// TIA Portal project "9230A V00 - PI" (V16)

(* hardware
DEVICE "S7-1200 station_1"  S7-1200 Station
   slot 0: "Rack_0"  S7-1200 Rack  Rack  V1.0
   slot 1: "1U2"  CPU 1212C DC/DC/DC  6ES7 212-1AE40-0XB0  V4.4
   slot 2: "2U2"  SM 1222 DQ8 x 24VDC  6ES7 222-1BF32-0XB0  V2.0
DEVICE "GSD device_1"  GSD.Device.PN
   slot 0: "Rack"  Rack  V1.0
   slot 0: "8DI"  8DI
   slot 0: "8DO"  8DO
   slot 0: "8DO"  8DO
   slot 0: "4AI, INT16[4] I"  4AI, INT16[4] I
   slot 0: "1U1"  750-375 V02.05.xx (FW 08)  750-375  V02.05.xx (08)
      slot 0: "Big Endian (MOTOROLA), Subslot-controlled PROFIenergy"  Big Endian (MOTOROLA), Subslot-controlled PROFIenergy
      slot 1: "Interface"  Interface
         slot 1: "Port 1"  Port 1
         slot 2: "Port 2"  Port 2
   slot 1: "2U1"  75x-430(/0..-...) 8DI  75x-430
   slot 2: "3U1"  75x-530(/0..-...) 8DO  75x-530
   slot 3: "4U1"  75x-530(/0..-...) 8DO  75x-530
   slot 4: "5U1"  75x-455(/0..-000) 4AI 4-20 mA s.e.  75x-455(/0..-000)
DEVICE "GSD device_2"  GSD.Device.PN
   slot 0: "Rack"  Rack  V1.0
   slot 0: "4AI, INT16[4] I"  4AI, INT16[4] I
   slot 0: "8DI"  8DI
   slot 0: "8DO"  8DO
   slot 0: "1U3"  750-375 V02.05.xx (FW 08)  750-375  V02.05.xx (08)
      slot 0: "Big Endian (MOTOROLA), Subslot-controlled PROFIenergy"  Big Endian (MOTOROLA), Subslot-controlled PROFIenergy
      slot 1: "Interface"  Interface
         slot 1: "Port 1"  Port 1
         slot 2: "Port 2"  Port 2
   slot 1: "2U3"  75x-430(/0..-...) 8DI  75x-430
   slot 2: "3U3"  75x-530(/0..-...) 8DO  75x-530
   slot 3: "4U3"  75x-455(/0..-000) 4AI 4-20 mA s.e.  75x-455(/0..-000)
DEVICE "SINAMICS G_1"  Sinamics.Device
   slot 0: "	_0"  Rail  SinamicsG120CRackP
   slot 0: "43G1"  G120C PN  6SL3210-1KE12-3UF2  4.7.10
      slot 1: "PROFINET interface"  MDD-SinamicsG120-P
      slot 3: "PM G120C"  PM G120C  6SL3210-1KE12-3UF2  -
DEVICE "SINAMICS G_2"  Sinamics.Device
   slot 0: "	_0"  Rail  SinamicsG120CRackP
   slot 0: "62G1"  G120C PN  6SL3210-1KE14-3UF2  4.7.10
      slot 1: "PROFINET interface"  MDD-SinamicsG120-P
      slot 3: "PM G120C"  PM G120C  6SL3210-1KE14-3UF2  -
DEVICE "SINAMICS G_3"  Sinamics.Device
   slot 0: "	_0"  Rail  SinamicsG120CRackP
   slot 0: "65G1"  G120C PN  6SL3210-1KE15-8UF2  4.7.10
      slot 1: "PROFINET interface"  MDD-SinamicsG120-P
      slot 3: "PM G120C"  PM G120C  6SL3210-1KE15-8UF2  -
DEVICE "SCALANCE X005"  SCALANCE X-Station
   slot 0: "SCALANCE X rack"  Rail
   slot 0: "Switch"  6GK5 008-0BA10-1AB2  V1.0
*)

// ===== PLC "1U2"  CPU 1212C DC/DC/DC =====

VAR_GLOBAL   // PLC tag table "Default tag table"
   "System_Byte" AT %MB1 : Byte;
   "FirstScan" AT %M1.0 : Bool;
   "DiagStatusUpdate" AT %M1.1 : Bool;
   "AlwaysTRUE" AT %M1.2 : Bool;
   "AlwaysFALSE" AT %M1.3 : Bool;
   "Clock_10Hz" AT %M0.0 : Bool;
   "Clock_5Hz" AT %M0.1 : Bool;
   "Clock_2.5Hz" AT %M0.2 : Bool;
   "Clock_2Hz" AT %M0.3 : Bool;
   "Clock_1.25Hz" AT %M0.4 : Bool;
   "Clock_1Hz" AT %M0.5 : Bool;
   "Clock_0.625Hz" AT %M0.6 : Bool;
   "Clock_0.5Hz" AT %M0.7 : Bool;
   "Clock_Byte" AT %MB0 : Byte;
   "Emergencia_Painel_1" AT %M7.5 : Bool;
   "Emergencia_Painel_3" AT %M7.6 : Bool;
   "Emergencia_Painel_2" AT %M7.7 : Bool;
END_VAR

VAR_GLOBAL   // PLC tag table "IO PAINEL 1"
   "EMERGENCIA_GERAL_PAINEL_1" AT %I1.0 : Bool;
   "NIVEL_SUPERIOR_SILO_2" AT %I1.1 : Bool;
   "SENSOR_23_POSICAO_1" AT %I1.2 : Bool;
   "NIVEL_INFERIOR_SILO_1" AT %I1.3 : Bool;
   "NIVEL_INFERIOR_SILO_2" AT %I1.5 : Bool;
   "SENSOR_23_POSICAO_2" AT %I1.4 : Bool;
   "NIVEL_SUPERIOR_SILO_1" AT %I1.6 : Bool;
   "BT_27_DOSAGEM_MANUAL" AT %I1.7 : Bool;
   "LIGA_LED_BT_27_DOSAGEM_MANUAL" AT %Q1.1 : Bool;
   "LIGA_22" AT %Q1.2 : Bool;
   "LIGA_26_SILO1_SENTIDO_1" AT %Q1.3 : Bool;
   "LIGA_23_SENTIDO_1" AT %Q1.4 : Bool;
   "LIGA_26_SILO1_SENTIDO_2" AT %Q1.5 : Bool;
   "LIGA_23_SENTIDO_2" AT %Q1.6 : Bool;
   "LIGA_26_SILO2_SENTIDO_1" AT %Q1.7 : Bool;
   "LIGA_26_SILO2_SENTIDO_2" AT %Q2.0 : Bool;
   "TARA_BALANCA_DOSAGEM" AT %Q2.1 : Bool;
   "LIGA_29" AT %Q2.2 : Bool;
   "LIGA_30" AT %Q2.4 : Bool;
   "ZERO_BALANCA_DOSAGEM" AT %Q2.6 : Bool;
   "POSICAO_ATUAL_26_SILO1" AT %IW68 : Int;
   "POSICAO_ATUAL_26_SILO2" AT %IW72 : Int;
   "PESO_ATUAL_DOSAGEM" AT %IW70 : Int;
END_VAR

VAR_GLOBAL   // PLC tag table "IO PAINEL 2"
   "LIGA_48" AT %Q8.0 : Bool;
   "LIGA_49_SENTIDO_1" AT %Q8.1 : Bool;
   "LIGA_49_SENTIDO_2" AT %Q8.2 : Bool;
   "CORRENTE_ATUAL_44" AT %IW64 : Int;
   "EMERGENCIA_GERAL_PAINEL_2" AT %I0.0 : Bool;
   "FALTA_FASE" AT %I0.1 : Bool;
   "NIVEL_INFERIOR_PRE_MISTURADOR" AT %I0.2 : Bool;
   "NIVEL_INFERIOR_POS_MISTURADOR" AT %I0.3 : Bool;
   "SENSOR_49_SENTIDO_1" AT %I0.4 : Bool;
   "SENSOR_49_SENTIDO_2" AT %I0.5 : Bool;
   "LIGA_42" AT %Q0.0 : Bool;
   "LIGA_CONTATOR_1_44" AT %Q0.1 : Bool;
   "LIGA_CONTATOR_2_44" AT %Q0.2 : Bool;
   "LIGA_44" AT %Q0.3 : Bool;
   "LIGA_45" AT %Q0.4 : Bool;
   "LIGA_46" AT %Q0.5 : Bool;
END_VAR

VAR_GLOBAL   // PLC tag table "IO PAINEL 3"
   "PESO_ATUAL_ENSAQUE" AT %IW76 : Int;
   "TARA_BALANCA_ENSAQUE" AT %Q3.2 : Bool;
   "ZERO_BALANCA_ENSAQUE" AT %Q3.0 : Bool;
   "EMERGENCIA_GERAL_PAINEL_3" AT %I2.0 : Bool;
   "NIVEL_SUPERIOR_SILO_EXP" AT %I2.2 : Bool;
   "NIVEL_INFERIOR_SILO_EXP" AT %I2.4 : Bool;
   "PEDAL_ENSAQUE" AT %I2.6 : Bool;
END_VAR

VAR_GLOBAL   // PLC tag table "teste"
   "TESTE" AT %MW16 : Int;
   "TESTE1" AT %MD12 : Real;
   "TESTE2" AT %MD8 : Real;
   "TESTE3" AT %M6.0 : Bool;
   "TESTE33" AT %MD2 : Real;
   "teste22" AT %MD18 : Real;
   "teste333" AT %MD22 : Real;
   "teste444" AT %MD26 : Real;
   "teste55" AT %MD30 : Real;
   "teste66" AT %M6.1 : Bool;
   "teste777" AT %M6.2 : Bool;
   "asdff" AT %M6.3 : Bool;
   "fdvxc" AT %M6.4 : Bool;
   "nhgfbvdc" AT %M6.5 : Bool;
   "teste123" AT %M6.7 : Bool;
   "tesdfsfdg" AT %M6.6 : Bool;
   "sdfvxc" AT %M7.0 : Bool;
   "teste88" AT %M7.1 : Bool;
   "teste99" AT %M7.2 : Bool;
   "teste00" AT %M7.3 : Bool;
   "teste3333" AT %M7.4 : Bool;
   "teste11" AT %M34.0 : Bool;
   "teste12" AT %M34.1 : Bool;
   "teste13" AT %M34.2 : Bool;
   "dfdfgsfgd" AT %M34.3 : Bool;
   "hngfnbfgn" AT %M34.4 : Bool;
   "teste411" AT %M34.5 : Bool;
   "teste412" AT %M34.6 : Bool;
END_VAR

TYPE "typeAtuadorLinearDigital"
   STRUCT
      Manual : Bool;   // em manual
      Automatico : Bool;   // em automatico
      Manutencao : Bool;   // em manutencao
      Libera_Bloqueio_Manual : Bool;   // Libera Bloqueio do motor
      Em_Emergencia : Bool;   // Em emergencia
      Liberado : Bool;   // Liberado
      Aciona_Lado1 : Bool;   // Comando aciona Lado
      Aciona_Lado2 : Bool;   // Comando aciona Lado
      Acionando_Lado1 : Bool;   // status acionando lado
      Acionando_Lado2 : Bool;   // status acionando lado
      Acionando_Automatico : Bool;   // acionando em modo automatico
      Em_Posicao_Lado1 : Bool;   // status lado atual
      Em_Posicao_Lado2 : Bool;   // status lado atual
      Falha_Acionando_Lado1 : Bool;   // falha acionando lado 1
      Falha_Acionando_Lado2 : Bool;   // falha acionando lado 2
      Falha_2_Posicoes_Ativa : Bool;   // falha quando os dois sensores estiverem ativos
      Falha_Confirmacao_Contator_Lado1 : Bool;   // falha no contator ou fio de confirmação do lado 1
      Falha_Confirmacao_Contator_Lado2 : Bool;   // falha no contator ou fio de confirmação do lado 2
      Reset_Falha : Bool;   // reset falha
      bitReserva : Bool;
      bitReserva_1 : Bool;
      bitReserva_2 : Bool;
      bitReserva_3 : Bool;
      bitReserva_4 : Bool;
      bitReserva_5 : Bool;
      bitReserva_6 : Bool;
      bitReserva_7 : Bool;
      bitReserva_8 : Bool;
      bitReserva_9 : Bool;
      bitReserva_10 : Bool;
      bitReserva_11 : Bool;
      bitReserva_12 : Bool;
   END_STRUCT;
END_TYPE

TYPE "typeAtuadorLinearAnalogico"
   STRUCT
      Liga_Manual : Bool;   // Liga/Desliga em manual
      Manual : Bool;   // em manual
      Automatico : Bool;   // em automatico
      Manutencao : Bool;   // em manutencao
      Libera_Bloqueio_Manual : Bool;   // Libera Bloqueio do motor
      Em_Emergencia : Bool;   // Em emergencia
      Liberado : Bool;   // Liberado
      Acionando_Automatico : Bool;   // acionando em modo automatico
      Falha_Confirmacao_Contator_Lado1 : Bool;   // falha no contator ou fio de confirmação do lado 1
      Falha_Confirmacao_Contator_Lado2 : Bool;   // falha no contator ou fio de confirmação do lado 2
      Falha_Posicionamento : Bool;   // falha de posicionamento entre a posicação atual e a posição solicitada
      Falha_Leitura_Posicao : Bool;   // falha de leitura de posição
      Reset_Falha : Bool;   // reset falha
      Aciona_Lado1 : Bool;   // Aciona lado 1 registro
      Aciona_Lado2 : Bool;   // Aciona lado 2 registro
      bitReserva_2 : Bool;
      bitReserva_3 : Bool;
      bitReserva_4 : Bool;
      bitReserva_5 : Bool;
      bitReserva_6 : Bool;
      bitReserva_7 : Bool;
      bitReserva_8 : Bool;
      bitReserva_9 : Bool;
      bitReserva_10 : Bool;
      bitReserva_11 : Bool;
      bitReserva_12 : Bool;
      bitReserva_13 : Bool;
      bitReserva_14 : Bool;
      bitReserva_15 : Bool;
      bitReserva_16 : Bool;
      bitReserva_17 : Bool;
      bitReserva_18 : Bool;
      Posicao_Solicitada_Automatico : Real;   // posicao solicita de 0 - 100%
      SP_Posicao_Manual : Real;   // Setpoint de posição manual
      Posicao_Atual : Real;   // posicao atual do atuador de 0 - 100%
   END_STRUCT;
END_TYPE

TYPE "typePD"
   STRUCT
      ligaManual : Bool;   // 0 = Desligar em modo Manual 1 = Ligar em modo Manual
      manual : Bool;
      automatico : Bool;
      manutencao : Bool;
      Libera_Bloqueio_Manual : Bool;
      reset : Bool;
      ligado : Bool;
      ligando : Bool;
      desligando : Bool;
      liberado : Bool;
      falhaPartidaNaoConfirmou : Bool;
      falhaContatorDesligou : Bool;
      falhaDisjuntoDesligou : Bool;
      falhaPartidaNaoDesligou : Bool;
      resetHotimetroTotal : Bool;
      resetHorimetroParcial : Bool;
      emergencia : Bool;
      disjuntorDesligado : Bool;
      tempoManutencao : Bool;
      falhaGeral : Bool;
      bitReserva : Bool;
      bitReserva_1 : Bool;
      bitReserva_2 : Bool;
      bitReserva_3 : Bool;
      bitReserva_4 : Bool;
      bitReserva_5 : Bool;
      bitReserva_6 : Bool;
      bitReserva_7 : Bool;
      bitReserva_8 : Bool;
      bitReserva_9 : Bool;
      bitReserva_10 : Bool;
      bitReserva_11 : Bool;
      SP_Manutencao : DInt;
      HorimetroParcial : DInt;
      HorimetroTotal : DInt;
      Tempo_Limpeza : DInt;
   END_STRUCT;
END_TYPE

TYPE "typeINV"
   STRUCT
      ligaManual : Bool;   // 0 = Desligar em modo Manual 1 = Ligar em modo Manual
      manual : Bool;
      automatico : Bool;
      manutencao : Bool;
      Libera_Bloqueio_Manual : Bool;
      reset : Bool;
      ligado : Bool;
      ligando : Bool;
      desligando : Bool;
      liberado : Bool;
      resetHotimetroTotal : Bool;
      resetHorimetroParcial : Bool;
      emergencia : Bool;
      disjuntorDesligado : Bool;
      tempoManutencao : Bool;
      falha : Bool;
      bitReserva : Bool;
      bitReserva_1 : Bool;
      bitReserva_2 : Bool;
      bitReserva_3 : Bool;
      bitReserva_4 : Bool;
      bitReserva_5 : Bool;
      bitReserva_6 : Bool;
      bitReserva_7 : Bool;
      bitReserva_8 : Bool;
      bitReserva_9 : Bool;
      bitReserva_10 : Bool;
      bitReserva_11 : Bool;
      bitReserva_12 : Bool;
      bitReserva_13 : Bool;
      bitReserva_14 : Bool;
      bitReserva_15 : Bool;
      Velocidade_Manual : Real;
      Velocidade_Automatica_Solicitada : Real;
      Velocidade_Atual : Real;
      Velocidade_Nominal : Real := 1800.0;
      SP_Corrente_Motor_Vazio : Real;
      Corrente_Atual : Real;
      Codigo_Alarme : Real;
      Codigo_Falha : Real;
      SP_Manutencao : DInt;
      HorimetroParcial : DInt;
      HorimetroTotal : DInt;
      Tempo_Limpeza : DInt;
   END_STRUCT;
END_TYPE

TYPE "typeSS"
   STRUCT
      ligaManual : Bool;   // 0 = Desligar em modo Manual 1 = Ligar em modo Manual
      manual : Bool;
      automatico : Bool;
      manutencao : Bool;
      Libera_Bloqueio_Manual : Bool;
      reset : Bool;
      ligado : Bool;
      ligando : Bool;
      desligando : Bool;
      liberado : Bool;
      falhaPartidaConfirmou : Bool;
      falhaContatorDesligou : Bool;
      falhaDisjuntoDesligou : Bool;
      falhaPartidaNaoDesligou : Bool;
      resetHotimetroTotal : Bool;
      resetHorimetroParcial : Bool;
      emergencia : Bool;
      disjuntorDesligado : Bool;
      tempoManutencao : Bool;
      falhaGeral : Bool;
      inverterSentidoGiro : Bool;
      SentidoGiro : Bool;   // 0 = Sentido 1, 1 = Sentido 2
      bitReserva : Bool;
      bitReserva_1 : Bool;
      bitReserva_2 : Bool;
      bitReserva_3 : Bool;
      bitReserva_4 : Bool;
      bitReserva_5 : Bool;
      bitReserva_6 : Bool;
      bitReserva_7 : Bool;
      bitReserva_8 : Bool;
      bitReserva_9 : Bool;
      SP_Manutencao : DInt;
      HorimetroParcial : DInt;
      HorimetroTotal : DInt;
      Tempo_Limpeza : DInt;
      Corrente_Atual : Real;
      SP_Corrente_Motor_Vazio : Real;
      SP_Tempo_Reversao : DInt := 1;   // Minutos Não pode ser menor que 1
      Tempo_Reversao_Atual : DInt;   // Minutos
   END_STRUCT;
END_TYPE

// folder: Chamadas/IDB/Controle Auto

DATA_BLOCK "IDB_Controle_Automatico"   // DB19
{ S7_Optimized_Access := 'TRUE' }
VERSION : 0.1
// stored: InstanceOfName Controle_Automatico
"Controle_Automatico"
BEGIN
END_DATA_BLOCK

DATA_BLOCK "Liga_Desl_Transporte_Pre_Mistura"   // DB24
{ S7_Optimized_Access := 'TRUE' }
VERSION : 0.1
// stored: InstanceOfName Liga_Desl_Sequencia
"Liga_Desl_Sequencia"
BEGIN
END_DATA_BLOCK

DATA_BLOCK "Liga_Desl_Moagem_Pos_Mistura"   // DB26
{ S7_Optimized_Access := 'TRUE' }
VERSION : 0.1
// stored: InstanceOfName Liga_Desl_Sequencia
"Liga_Desl_Sequencia"
BEGIN
END_DATA_BLOCK

DATA_BLOCK "Liga_Desl_Transporte_Produto_Acabado"   // DB27
{ S7_Optimized_Access := 'TRUE' }
VERSION : 0.1
// stored: InstanceOfName Liga_Desl_Sequencia
"Liga_Desl_Sequencia"
BEGIN
END_DATA_BLOCK

// folder: Chamadas/IDB/Equipamentos

DATA_BLOCK "IDB_23"   // DB1
{ S7_Optimized_Access := 'TRUE' }
VERSION : 0.1
// stored: InstanceOfName Atuador_Linear_Bifurcada
"Atuador_Linear_Bifurcada"
BEGIN
END_DATA_BLOCK

DATA_BLOCK "IDB_22"   // DB3
{ S7_Optimized_Access := 'TRUE' }
VERSION : 0.1
// stored: InstanceOfName PD
"PD"
BEGIN
END_DATA_BLOCK

DATA_BLOCK "IDB_29"   // DB4
{ S7_Optimized_Access := 'TRUE' }
VERSION : 0.1
// stored: InstanceOfName PD
"PD"
BEGIN
END_DATA_BLOCK

DATA_BLOCK "IDB_30"   // DB5
{ S7_Optimized_Access := 'TRUE' }
VERSION : 0.1
// stored: InstanceOfName PD
"PD"
BEGIN
END_DATA_BLOCK

DATA_BLOCK "IDB_42"   // DB6
{ S7_Optimized_Access := 'TRUE' }
VERSION : 0.1
// stored: InstanceOfName PD
"PD"
BEGIN
END_DATA_BLOCK

DATA_BLOCK "IDB_43"   // DB7
{ S7_Optimized_Access := 'TRUE' }
VERSION : 0.1
// stored: InstanceOfName INV
"INV"
BEGIN
END_DATA_BLOCK

DATA_BLOCK "IDB_44"   // DB8
{ S7_Optimized_Access := 'TRUE' }
VERSION : 0.1
// stored: InstanceOfName SS_MOINHO
"SS_MOINHO"
BEGIN
END_DATA_BLOCK

DATA_BLOCK "IDB_45"   // DB9
{ S7_Optimized_Access := 'TRUE' }
VERSION : 0.1
// stored: InstanceOfName PD
"PD"
BEGIN
END_DATA_BLOCK

DATA_BLOCK "IDB_46"   // DB10
{ S7_Optimized_Access := 'TRUE' }
VERSION : 0.1
// stored: InstanceOfName PD
"PD"
BEGIN
END_DATA_BLOCK

DATA_BLOCK "IDB_48"   // DB11
{ S7_Optimized_Access := 'TRUE' }
VERSION : 0.1
// stored: InstanceOfName PD
"PD"
BEGIN
END_DATA_BLOCK

DATA_BLOCK "IDB_62"   // DB12
{ S7_Optimized_Access := 'TRUE' }
VERSION : 0.1
// stored: InstanceOfName INV
"INV"
BEGIN
END_DATA_BLOCK

DATA_BLOCK "IDB_65"   // DB13
{ S7_Optimized_Access := 'TRUE' }
VERSION : 0.1
// stored: InstanceOfName INV
"INV"
BEGIN
END_DATA_BLOCK

DATA_BLOCK "IDB_26_SILO1"   // DB16
{ S7_Optimized_Access := 'TRUE' }
VERSION : 0.1
// stored: InstanceOfName Atuador_Linear_Analogico
"Atuador_Linear_Analogico"
BEGIN
END_DATA_BLOCK

DATA_BLOCK "IDB_26_SILO2"   // DB17
{ S7_Optimized_Access := 'TRUE' }
VERSION : 0.1
// stored: InstanceOfName Atuador_Linear_Analogico
"Atuador_Linear_Analogico"
BEGIN
END_DATA_BLOCK

DATA_BLOCK "IDB_49"   // DB18
{ S7_Optimized_Access := 'TRUE' }
VERSION : 0.1
// stored: InstanceOfName Atuador_Linear_Digital
"Atuador_Linear_Digital"
BEGIN
END_DATA_BLOCK

// folder: DB

DATA_BLOCK "DB_Controle_Automatico"   // DB20
{ S7_Optimized_Access := 'TRUE' }
VERSION : 0.1
   VAR RETAIN
      Controle : Struct
         Dosagem_Materia_Prima : Struct
            Ligar : Bool;   // Solicita ligar Dosagem
            Ligado : Bool;   // Dosagem Ligada
            Liberado_Nova_Dosagem : Bool;   // Liberado dosagem de nova batelada
            Finalizado_Dosagem : Bool;   // finalizado dosagem da batelada solicitada
            Balanca_Vazia : Bool;   // Solicita balança vazia
            Habilita_Setar_Balanca_Vazia : Bool;   // habilita solicitar balança vazia
            Reserva : Bool;
            Reserva_1 : Bool;
            Passo_Atual : Int;   // Passo Atual da dosagem
            Dosagem_Materia_Prima_Silo_1 : Real;   // Valor em Kg da dosagem de materia prima do silo 1 solicitada
            Dosagem_Materia_Prima_Silo_2 : Real;   // Valor em Kg da dosagem de materia prima do silo 2 solicitada
            Dosado_Materia_Prima_Silo_1 : Real;   // Valor dosado do silo 1 na balança
            Dosado_Materia_Prima_Silo_2 : Real;   // Valor dosado do silo 2 na balança
            Complemento_Pre : Struct   // Complementos dosados manualmente na balança
               Quantidade_Itens : Int;   // Quantidade de complementos na receita
               Item_Atual : Int;   // Em qual item da receita esta no momento
               Quantidade_Dosada_Item_Atual : Real;   // Quantidade dosada do item atual, valor disponível após finalizado dosagem
               Habilitado_Inicio_Dosagem : Bool;   // Habilita o inicio da dosagem manual
               Botao_Inicio_Fim_Dosagem_IHM : Bool;   // Bit para iniciar ou finalizar dosagem pela IHM
               Item_Atual_Iniciado_Dosagem : Bool;   // Se iniciou a dosagem do item atual
               Item_Atual_Finalizado_Dosagem : Bool;   // Se finalizou a dosagem do item atual
               Finalizado_Dosagem_Complementos : Bool;   // Se finalizou a dosagem de todos os complementos
               Reserva : Bool;
               Reserva_1 : Bool;
               Reserva_2 : Bool;
            END_STRUCT;
         END_STRUCT;
         Transporte_Para_Pre_Mistura : Struct
            Ligar : Bool;   // Solicita ligar transporte
            Ligado : Bool;   // Transporte ligado
            Liberado_Iniciar_Transporte : Bool;   // liberado iniciar transporte
            Reserva : Bool;
            Reserva_1 : Bool;
            Reserva_2 : Bool;
            Reserva_3 : Bool;
            Reserva_4 : Bool;
         END_STRUCT;
         Pre_Mistura : Struct
            Ligar : Bool;   // Solicita ligar pré mistura
            Ligado : Bool;   // Pré mistura ligado
            Liberado_Nova_Batelada : Bool;   // Liberado mistura de nova batelada
            Recebendo_Produto : Bool;   // Esta recebendo produto
            Iniciado_Mistura : Bool;   // Iniciado a mistura
            Finalizado_Mistura : Bool;   // Finalizado mistura
            Reserva : Bool;
            Reserva_1 : Bool;
            Tempo_SP : DInt;   // Tempo em segundos de mistura
            Tempo_Restante : DInt;   // Tempo em segundos restante
         END_STRUCT;
         Moagem_Pos_Mistura : Struct
            Ligar : Bool;   // Solicita ligar moagem
            Ligado : Bool;   // Moagem ligado
            Liberado_Nova_Moagem : Bool;   // Liberado moagem de nova batelada
            Finalizou_Moagem : Bool;   // Finalizou Moagem
            Reserva : Bool;
            Reserva_1 : Bool;
            Reserva_2 : Bool;
            Reserva_3 : Bool;
         END_STRUCT;
         Pos_Mistura : Struct
            Ligar : Bool;   // Solicita ligar pós mistura
            Ligado : Bool;   // pós mistura ligado
            Liberado_Nova_Batelada : Bool;   // liberado mistura de nova batelada
            Recebendo_Produto : Bool;   // Esta recebendo produto
            Iniciado_Mistura : Bool;   // Iniciado a mistura
            Finalizado_Mistura : Bool;   // Finalizado mistura
            Reserva : Bool;
            Reserva_1 : Bool;
            Tempo_SP : DInt;   // Tempo em segundos de mistura
            Tempo_Restante : DInt;   // Tempo em segundos restante
            Complemento_Pos : Struct   // Complementos dosados manualmente na balança
               Quantidade_Itens : Int;   // Quantidade de complementos na receita
               Item_Atual : Int;   // Em qual item da receita esta no momento
               Quantidade_Dosada_Item_Atual : Real;   // Quantidade dosada do item atual, valor disponível após finalizado dosagem
               Habilitado_Inicio_Dosagem : Bool;   // Habilita o inicio da dosagem manual
               Botao_Inicio_Fim_Dosagem_IHM : Bool;   // Bit para iniciar ou finalizar dosagem pela IHM
               Item_Atual_Iniciado_Dosagem : Bool;   // Se iniciou a dosagem do item atual
               Item_Atual_Finalizado_Dosagem : Bool;   // Se finalizou a dosagem do item atual
               Finalizado_Dosagem_Complementos : Bool;   // Se finalizou a dosagem de todos os complementos
               Reserva : Bool;
               Reserva_1 : Bool;
               Reserva_2 : Bool;
            END_STRUCT;
         END_STRUCT;
         Transporte_Produto_Acabado : Struct
            Ligar : Bool;   // Solicita ligar transporte para produto acabado
            Ligado : Bool;   // Transporte para produto acabado ligado
            Liberado_Iniciar_Transporte : Bool;   // Liberado transporte nova batelada para produto acabado
            Reserva : Bool;
            Reserva_1 : Bool;
            Reserva_2 : Bool;
            Reserva_3 : Bool;
            Reserva_4 : Bool;
         END_STRUCT;
      END_STRUCT;
   END_VAR
BEGIN
END_DATA_BLOCK

// folder: Supervisao

DATA_BLOCK "DB_Controle_Equip"   // DB2
{ S7_Optimized_Access := 'FALSE' }
VERSION : 0.1
   VAR
      "22" : "typePD";
      "23" : "typeAtuadorLinearDigital";
      "26_Silo1" : "typeAtuadorLinearAnalogico";
      "26_Silo2" : "typeAtuadorLinearAnalogico";
      "29" : "typePD";
      "30" : "typePD";
      "42" : "typePD";
      "43" : "typeINV";
      "44" : "typeSS";
      "45" : "typePD";
      "46" : "typePD";
      "48" : "typePD";
      "49" : "typeAtuadorLinearDigital";
      "62" : "typeINV";
      "65" : "typeINV";
   END_VAR
BEGIN
END_DATA_BLOCK

DATA_BLOCK "DB_Producao_Automatica"   // DB15
{ S7_Optimized_Access := 'FALSE' }
VERSION : 0.1
   VAR
      Controle : Struct
         Slot1_Batelada : Struct
            Tempo_Pre_Mistura : DInt;   // Tempo de pré Mistura
            Tempo_Pos_Mistura : DInt;   // Tempo de pós Mistura
            Peso_Total_Batelada_Desejado : Real;   // Peso total desejado da batelada
            Dosagem_Materia_Prima_Silo_1 : Real;   // Dosagem Materia Prima no Silo 1
            Dosagem_Materia_Prima_Silo_2 : Real;   // Dosagem Materia Prima no Silo 2
            Dosado_Materia_Prima_Silo_1 : Real;   // Dosado Materia Prima no Silo 1
            Dosado_Materia_Prima_Silo_2 : Real;   // Dosado Materia Prima no Silo 2
            Complemento_Pre : Struct   // Complemento ou Matéria Prima dosada manualmente na Balança
               Quantidade_Itens : Int;   // Qtd itens dosagem Manual
               Item_Atual : Int;   // Item atual
               Quantidade_Dosada_Item_Atual : Real;   // Qtd dosada item Atual
               Quantidade_Dosada_Total : Real;   // Qtd dosada Total
               Habilitado_Inicio_Dosagem : Bool;   // Habilita Iniciar a dosagem
               Botao_Inicio_Fim_Dosagem_IHM : Bool;   // BT Inicia ou finaliza Dosagem
               Item_Atual_Iniciado_Dosagem : Bool;   // Iniciado Dosagem item atual
               Item_Atual_Finalizado_Dosagem : Bool;   // Finalizado Dosagem item atual
               Finalizado_Dosagem_Complementos : Bool;   // Finalizado a dosagem de todos complementos
               Reserva : Bool;   // reserva
               Reserva_1 : Bool;   // reserva
               Reserva_2 : Bool;   // reserva
            END_STRUCT;
            Complemento_Pos : Struct   // Complemento ou Matéria Prima dosada manualmente na Pós Mistura
               Quantidade_Itens : Int;   // Qtd itens dosagem Manual
               Item_Atual : Int;   // Item atual
               Quantidade_Dosada_Item_Atual : Real;   // Qtd dosada item Atual
               Quantidade_Dosada_Total : Real;   // Qtd dosada Total
               Habilitado_Inicio_Dosagem : Bool;   // Habilita Iniciar a dosagem
               Botao_Inicio_Fim_Dosagem_IHM : Bool;   // BT Inicia ou finaliza Dosagem
               Item_Atual_Iniciado_Dosagem : Bool;   // Iniciado Dosagem item atual
               Item_Atual_Finalizado_Dosagem : Bool;   // Finalizado Dosagem item atual
               Finalizado_Dosagem_Complementos : Bool;   // Finalizado a dosagem de todos complementos
               Reserva : Bool;   // reserva
               Reserva_1 : Bool;   // reserva
               Reserva_2 : Bool;   // reserva
            END_STRUCT;
            TempoAtualDesdeIniciado : DInt;   // Tempo total desde iniciado a produção da batelada
            TempoAtualPasso : DInt;   // Tempo atual de cada passo, como tempo em dosagem manual, tempo em pré mistura...
            Status : Int;   // Status da batelada
            Command : Struct   // Palavra de comando do Slot
               Solicita_Nova_Batelada : Bool;   // Slot Disponível para iniciar nova Batelada
               Iniciou : Bool;   // Iniciou batelada
               Finalizou : Bool;   // finalizou batelada
               Carregou_Nova_Batelada : Bool;
               reserva_1 : Bool;
               reserva_2 : Bool;
               reserva_3 : Bool;
               reserva_4 : Bool;
               reserva_5 : Bool;
               reserva_6 : Bool;
               reserva_7 : Bool;
               reserva_8 : Bool;
               reserva_9 : Bool;
               reserva_10 : Bool;
               reserva_11 : Bool;
               reserva_12 : Bool;
               reserva_13 : Bool;
               reserva_14 : Bool;
               reserva_15 : Bool;
               reserva_16 : Bool;
               reserva_17 : Bool;
               reserva_18 : Bool;
               reserva_19 : Bool;
               reserva_20 : Bool;
               reserva_21 : Bool;
               reserva_22 : Bool;
               reserva_23 : Bool;
               reserva_24 : Bool;
               reserva_25 : Bool;
               reserva_26 : Bool;
               reserva_27 : Bool;
               reserva_28 : Bool;
            END_STRUCT;
         END_STRUCT;
         Bateladas_Iniciadas : Int;
         Bateladas_Finalizadas : Int;
         Command : Struct
            IniciarProducao : Bool;
            Habilitado_Iniciar_Nova_Producao : Bool;
            reserva_1 : Bool;
            reserva_2 : Bool;
            reserva_3 : Bool;
            reserva_4 : Bool;
            reserva_5 : Bool;
            reserva_6 : Bool;
            reserva_7 : Bool;
            reserva_8 : Bool;
            reserva_9 : Bool;
            reserva_10 : Bool;
            reserva_11 : Bool;
            reserva_12 : Bool;
            reserva_13 : Bool;
            reserva_14 : Bool;
            reserva_15 : Bool;
            reserva_16 : Bool;
            reserva_17 : Bool;
            reserva_18 : Bool;
            reserva_19 : Bool;
            reserva_20 : Bool;
            reserva_21 : Bool;
            reserva_22 : Bool;
            reserva_23 : Bool;
            reserva_24 : Bool;
            reserva_25 : Bool;
            reserva_26 : Bool;
            reserva_27 : Bool;
            reserva_28 : Bool;
            reserva_29 : Bool;
            reserva_30 : Bool;
         END_STRUCT;
      END_STRUCT;
   END_VAR
BEGIN
END_DATA_BLOCK

DATA_BLOCK "DB_PID"   // DB21
{ S7_Optimized_Access := 'TRUE' }
VERSION : 0.1
   VAR
      Moinho : Struct
         Habilita_PID : Bool;
         Reserva : Bool;
         Reserva_1 : Bool;
         Reserva_2 : Bool;
         Reserva_3 : Bool;
         Reserva_4 : Bool;
         Reserva_5 : Bool;
         Reserva_6 : Bool;
         SetPoint : Real;   // Setpoint Corrente
         Proporcional : Real;
         Integral : Real;
         Derivado : Real;
         Limite_Max : Real;
         Limite_Min : Real;
      END_STRUCT;
   END_VAR
BEGIN
END_DATA_BLOCK

DATA_BLOCK "DB_Auxiliares"   // DB22
{ S7_Optimized_Access := 'TRUE' }
VERSION : 0.1
   VAR
      NIVEIS : Struct
         SUPERIOR_SILO_1 : Bool;
         SUPERIOR_SILO_2 : Bool;
         SUPERIOR_SILO_EXP : Bool;
         INFERIOR_SILO_1 : Bool;
         INFERIOR_SILO_2 : Bool;
         INFERIOR_SILO_EXP : Bool;
         INFERIOR_PREMISTURADOR : Bool;
         INFERIOR_POSMISTURADOR : Bool;
         reserva_2 : Bool;
         reserva_3 : Bool;
         reserva_4 : Bool;
         reserva_5 : Bool;
         reserva_6 : Bool;
         reserva_7 : Bool;
         reserva_8 : Bool;
         reserva_9 : Bool;
         reserva_10 : Bool;
         reserva_11 : Bool;
         reserva_12 : Bool;
         reserva_13 : Bool;
         reserva_14 : Bool;
         reserva_15 : Bool;
         reserva_16 : Bool;
         reserva_17 : Bool;
         reserva_18 : Bool;
         reserva_19 : Bool;
         reserva_20 : Bool;
         reserva_21 : Bool;
         reserva_22 : Bool;
         reserva_23 : Bool;
         reserva_24 : Bool;
         reserva_25 : Bool;
      END_STRUCT;
   END_VAR
BEGIN
END_DATA_BLOCK

DATA_BLOCK "DB_Configuracoes"   // DB23
{ S7_Optimized_Access := 'FALSE' }
VERSION : 0.1
   VAR
      Maquinas : Struct
         Maximo_Silo_Produto_Acabado : Real;
         Maximo_Silo_1_Materia_Prima : Real;
         Maximo_Silo_2_Materia_Prima : Real;
         Maximo_Balanca : Real;
         Maximo_PreMisturador : Real;
         Maximo_PosMisturador : Real;
      END_STRUCT;
      Registro_26 : Struct
         Abertura_Maxima_Silo_1 : Real := 100.0;   // Percentual de abertura máximo do registro 26 Silo 1
         Inicio_Reducao_Silo_1 : Real := 70.0;   // Percentual do inicio da redução do registro 26 Silo 1
         Fechamento_Antecipado_Silo_1 : Real := 1.0;
         Abertura_Maxima_Silo_2 : Real := 100.0;   // Percentual de abertura máximo do registro 26 Silo 2
         Inicio_Reducao_Silo_2 : Real := 70.0;   // Percentual do inicio da redução do registro 26 Silo 2
         Fechamento_Antecipado_Silo_2 : Real := 1.0;
      END_STRUCT;
   END_VAR
BEGIN
END_DATA_BLOCK

// folder: (top level)

ORGANIZATION_BLOCK "Main"   // OB1, FBD, ProgramCycle
TITLE = "Main Program Sweep (Cycle)"
{ S7_Optimized_Access := 'TRUE' }
VERSION : 0.1
   VAR_INPUT
      Initial_Call : Bool;   // Initial call of this OB
      Remanence : Bool;   // =True, if remanent data are available
   END_VAR
BEGIN

REGION Network 1: Emergencia
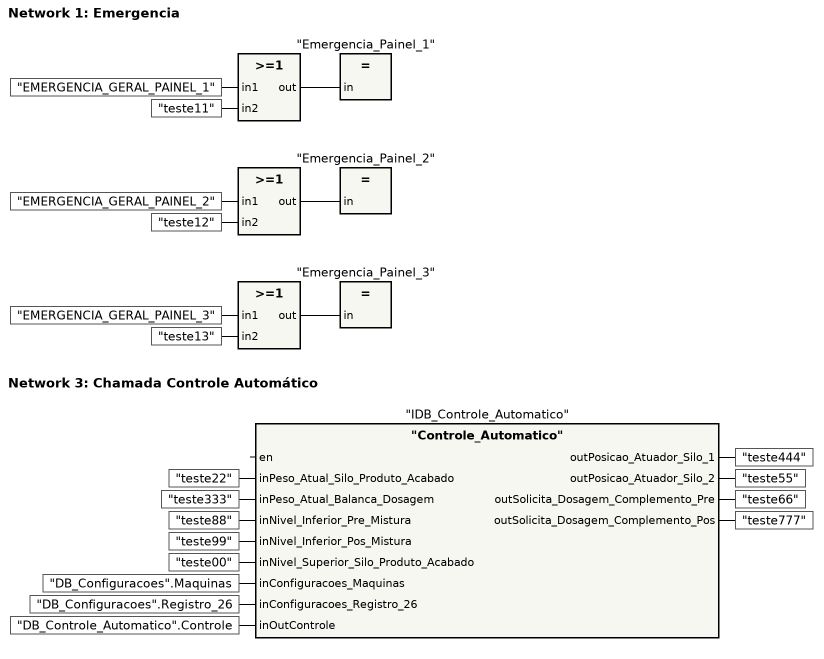
   "Emergencia_Painel_1" := "EMERGENCIA_GERAL_PAINEL_1" OR "teste11";
   "Emergencia_Painel_2" := "EMERGENCIA_GERAL_PAINEL_2" OR "teste12";
   "Emergencia_Painel_3" := "EMERGENCIA_GERAL_PAINEL_3" OR "teste13";
END_REGION

REGION Network 2: Chamada Controle Produção
END_REGION

REGION Network 3: Chamada Controle Automático
   "IDB_Controle_Automatico"(inPeso_Atual_Silo_Produto_Acabado := "teste22",   // "Controle_Automatico"
                           inPeso_Atual_Balanca_Dosagem := "teste333",
                           inNivel_Inferior_Pre_Mistura := "teste88",
                           inNivel_Inferior_Pos_Mistura := "teste99",
                           inNivel_Superior_Silo_Produto_Acabado := "teste00",
                           inConfiguracoes_Maquinas := "DB_Configuracoes".Maquinas,
                           inConfiguracoes_Registro_26 := "DB_Configuracoes".Registro_26,
                           inOutControle := "DB_Controle_Automatico".Controle,
                           outPosicao_Atuador_Silo_1 => "teste444",
                           outPosicao_Atuador_Silo_2 => "teste55",
                           outSolicita_Dosagem_Complemento_Pre => "teste66",
                           outSolicita_Dosagem_Complemento_Pos => "teste777");
END_REGION

REGION Network 4: Liga/ Desliga Automatico
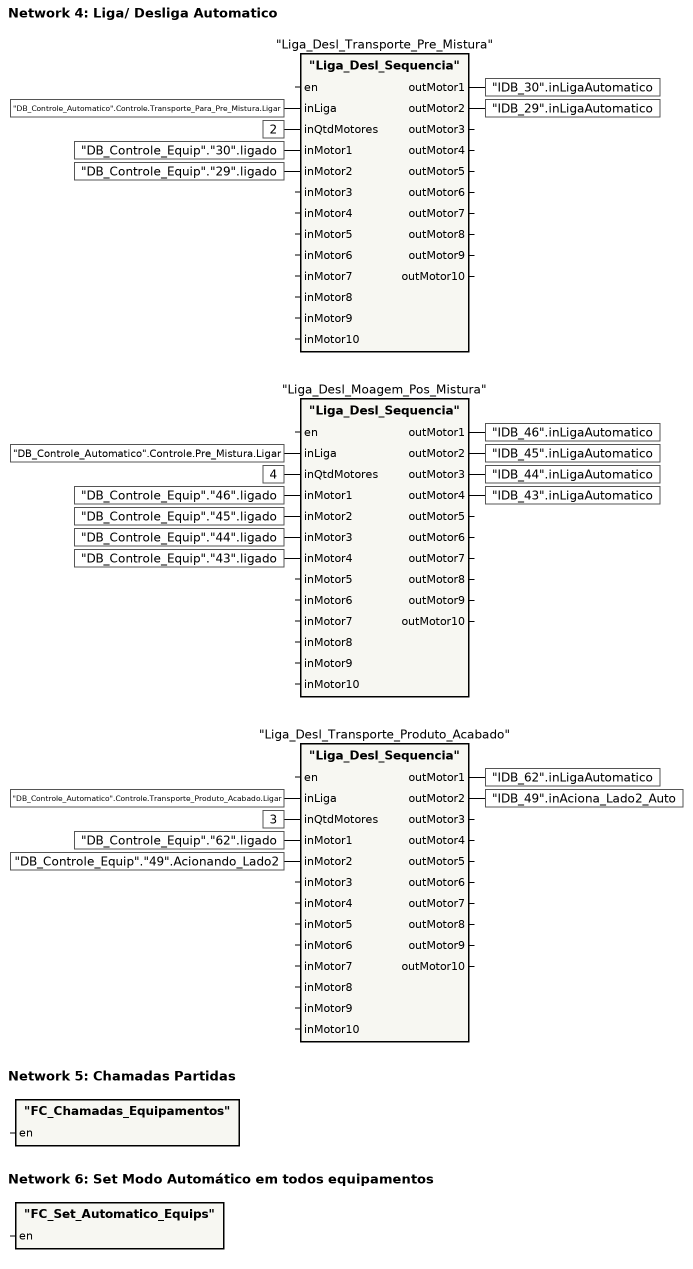
   "Liga_Desl_Transporte_Pre_Mistura"(inLiga := "DB_Controle_Automatico".Controle.Transporte_Para_Pre_Mistura.Ligar,   // "Liga_Desl_Sequencia": Liga e desliga Transporte para Pré Mistura
                           inQtdMotores := 2,
                           inMotor1 := "DB_Controle_Equip"."30".ligado,
                           inMotor2 := "DB_Controle_Equip"."29".ligado,
                           outMotor1 => "IDB_30".inLigaAutomatico,
                           outMotor2 => "IDB_29".inLigaAutomatico);
   "Liga_Desl_Moagem_Pos_Mistura"(inLiga := "DB_Controle_Automatico".Controle.Pre_Mistura.Ligar,   // "Liga_Desl_Sequencia": Liga e desliga Moagem
                           inQtdMotores := 4,
                           inMotor1 := "DB_Controle_Equip"."46".ligado,
                           inMotor2 := "DB_Controle_Equip"."45".ligado,
                           inMotor3 := "DB_Controle_Equip"."44".ligado,
                           inMotor4 := "DB_Controle_Equip"."43".ligado,
                           outMotor1 => "IDB_46".inLigaAutomatico,
                           outMotor2 => "IDB_45".inLigaAutomatico,
                           outMotor3 => "IDB_44".inLigaAutomatico,
                           outMotor4 => "IDB_43".inLigaAutomatico);
   "Liga_Desl_Transporte_Produto_Acabado"(inLiga := "DB_Controle_Automatico".Controle.Transporte_Produto_Acabado.Ligar,   // "Liga_Desl_Sequencia": Liga e desliga Transporte para produto acabdo
                           inQtdMotores := 3,
                           inMotor1 := "DB_Controle_Equip"."62".ligado,
                           inMotor2 := "DB_Controle_Equip"."49".Acionando_Lado2,
                           outMotor1 => "IDB_62".inLigaAutomatico,
                           outMotor2 => "IDB_49".inAciona_Lado2_Auto);
END_REGION

REGION Network 5: Chamadas Partidas
   "FC_Chamadas_Equipamentos"();
END_REGION

REGION Network 6: Set Modo Automático em todos equipamentos
   "FC_Set_Automatico_Equips"();
END_REGION
END_ORGANIZATION_BLOCK

ORGANIZATION_BLOCK "Cyclic interrupt"   // OB30, FBD, CyclicInterrupt
{ S7_Optimized_Access := 'TRUE' }
VERSION : 0.1
   VAR_INPUT
      Initial_Call : Bool;   // Initial call of this OB
      Event_Count : Int;   // Events discarded
   END_VAR
BEGIN

REGION Network 1
   // 43 É o alimentador do moinho
   // 44 é o motor do moinho
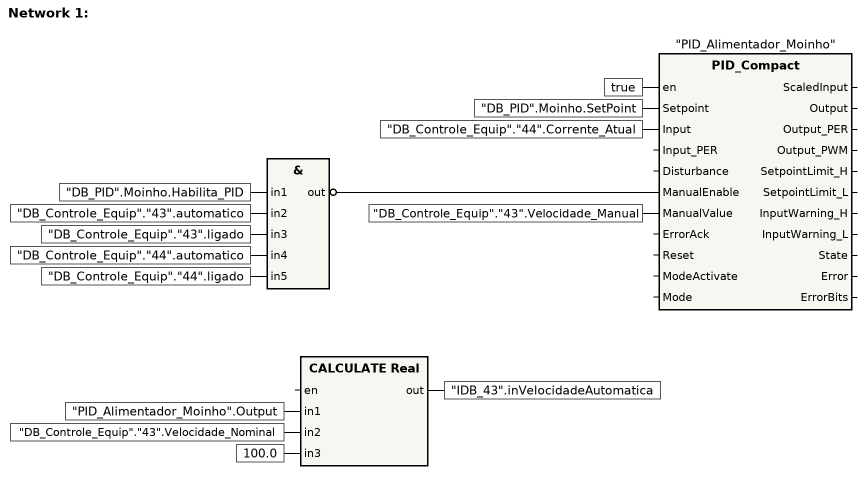
   IF true THEN
       "PID_Alimentador_Moinho"(Setpoint := "DB_PID".Moinho.SetPoint,   // PID_Compact
                               Input := "DB_Controle_Equip"."44".Corrente_Atual,
                               ManualEnable := NOT ("DB_PID".Moinho.Habilita_PID AND "DB_Controle_Equip"."43".automatico AND "DB_Controle_Equip"."43".ligado AND "DB_Controle_Equip"."44".automatico AND "DB_Controle_Equip"."44".ligado),
                               ManualValue := "DB_Controle_Equip"."43".Velocidade_Manual);
   END_IF;
   "IDB_43".inVelocidadeAutomatica := ("PID_Alimentador_Moinho".Output*"DB_Controle_Equip"."43".Velocidade_Nominal)/100.0;
END_REGION

REGION Network 2 (SCL)
   "PID_Alimentador_Moinho".Config.OutputUpperLimit := ("DB_PID".Moinho.Limite_Max * 100) / "DB_Controle_Equip"."43".Velocidade_Nominal;
   "PID_Alimentador_Moinho".Config.OutputLowerLimit := ("DB_PID".Moinho.Limite_Min * 100) / "DB_Controle_Equip"."43".Velocidade_Nominal;

   IF "PID_Alimentador_Moinho".ErrorBits <> 0 THEN
       "PID_Alimentador_Moinho".ErrorAck := true;
   END_IF;
END_REGION
END_ORGANIZATION_BLOCK

// folder: Chamadas

FUNCTION "FC_Chamadas_Equipamentos" : Void   // FC1, FBD
{ S7_Optimized_Access := 'TRUE' }
VERSION : 0.1
   VAR_TEMP   // added for the SCL form of the ladder/FBD networks
      _w1 : Bool;
   END_VAR
BEGIN

REGION Network 1 (SCL): NIVEIS
   //Níveis superiores
   "DB_Auxiliares".NIVEIS.SUPERIOR_SILO_1 := "NIVEL_SUPERIOR_SILO_1"; //24
   "DB_Auxiliares".NIVEIS.SUPERIOR_SILO_2 := "NIVEL_SUPERIOR_SILO_2"; //24
   "DB_Auxiliares".NIVEIS.SUPERIOR_SILO_EXP := "NIVEL_SUPERIOR_SILO_EXP"; //63

   //Níveis inferiories
   "DB_Auxiliares".NIVEIS.INFERIOR_SILO_1 := "NIVEL_INFERIOR_SILO_1";
   "DB_Auxiliares".NIVEIS.INFERIOR_SILO_2 := "NIVEL_INFERIOR_SILO_2";
   "DB_Auxiliares".NIVEIS.INFERIOR_SILO_EXP := "NIVEL_INFERIOR_SILO_EXP";
   "DB_Auxiliares".NIVEIS.INFERIOR_PREMISTURADOR := "NIVEL_INFERIOR_PRE_MISTURADOR";
   "DB_Auxiliares".NIVEIS.INFERIOR_POSMISTURADOR := "NIVEL_INFERIOR_POS_MISTURADOR";
END_REGION

REGION Network 2: PAINEL 1 ================================================================
END_REGION

REGION Network 3: 21 - ROSCA MP COM MOEGA ABASTECIMENTO MANUAL
END_REGION

REGION Network 4: 22 - ELEVADOR AUTOLIMPANTE MATERIA PRIMA
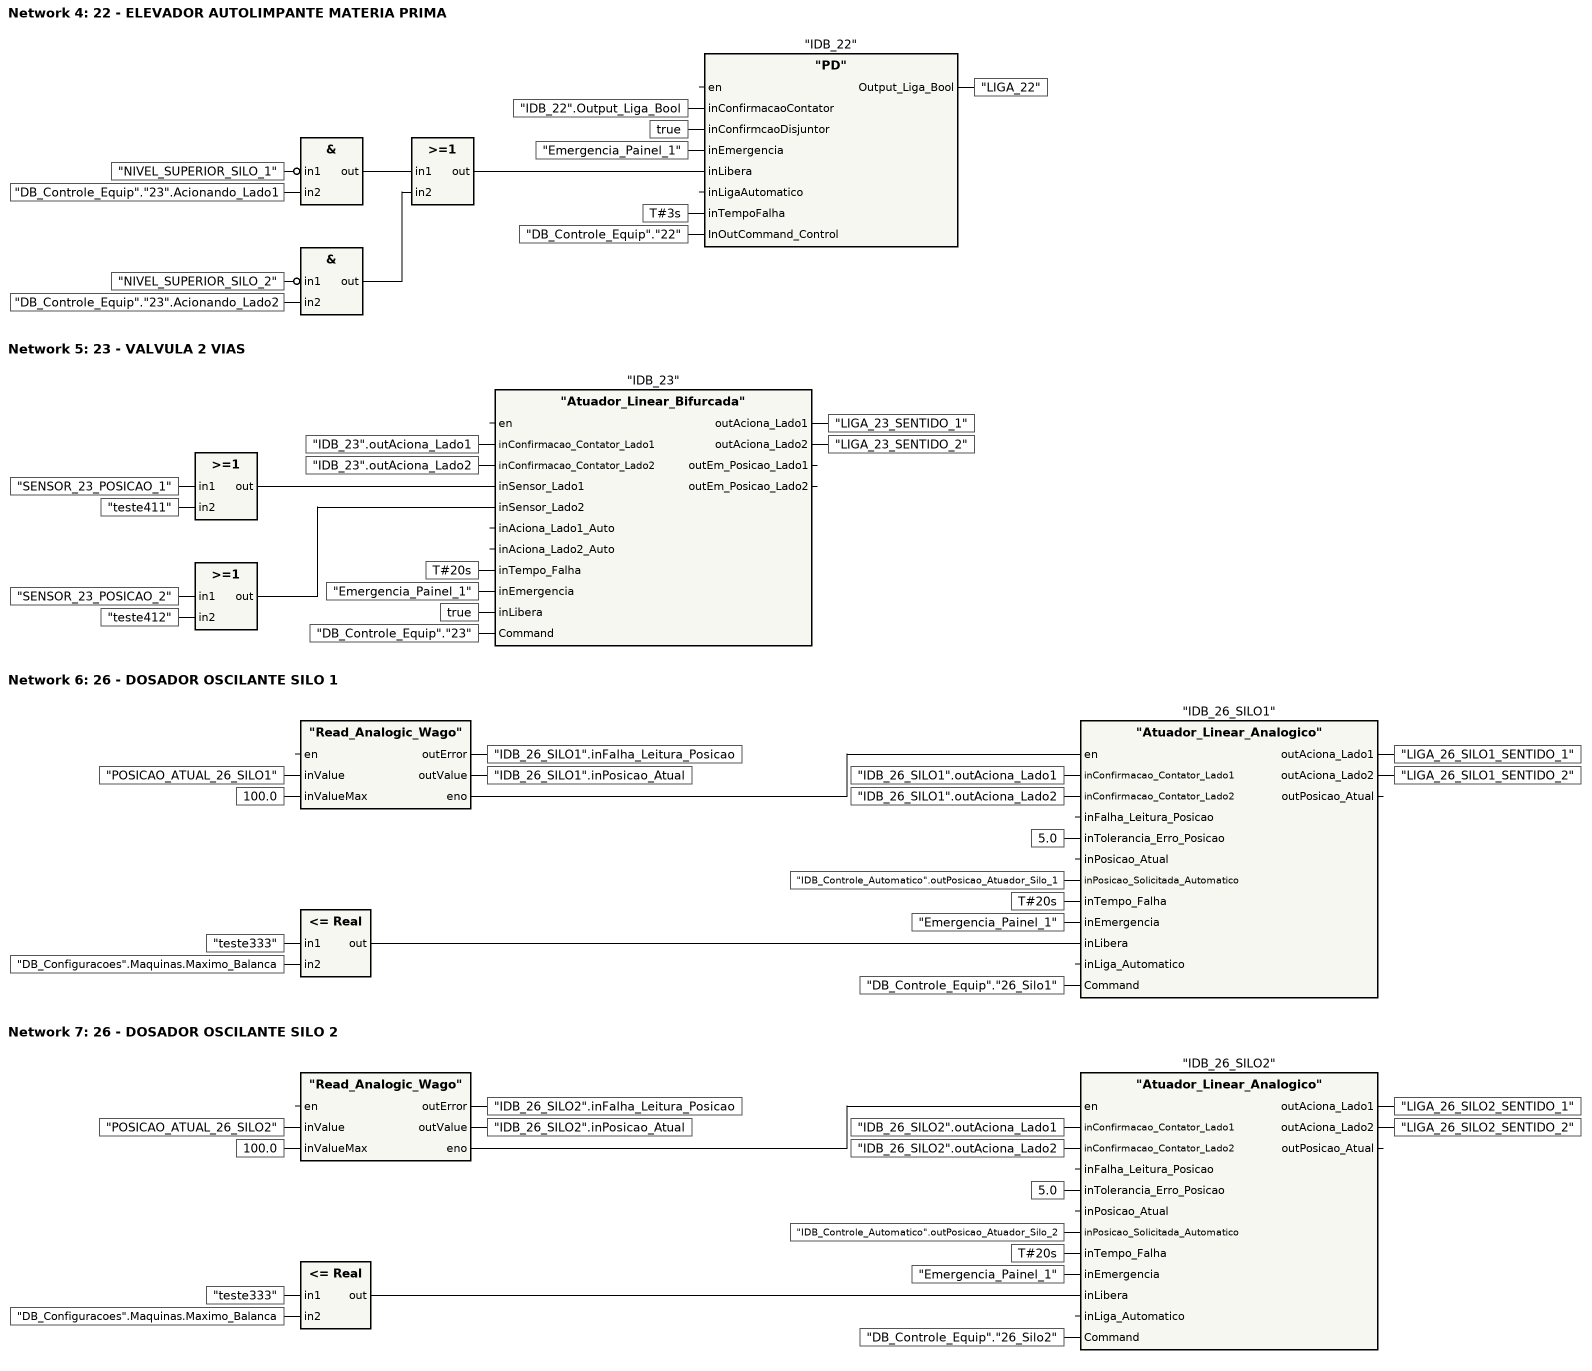
   "IDB_22"(inConfirmacaoContator := "IDB_22".Output_Liga_Bool,   // "PD"
            inConfirmcaoDisjuntor := true,
            inEmergencia := "Emergencia_Painel_1",
            inLibera := (NOT "NIVEL_SUPERIOR_SILO_1" AND "DB_Controle_Equip"."23".Acionando_Lado1) OR (NOT "NIVEL_SUPERIOR_SILO_2" AND "DB_Controle_Equip"."23".Acionando_Lado2),
            inTempoFalha := T#3s,
            InOutCommand_Control := "DB_Controle_Equip"."22",
            Output_Liga_Bool => "LIGA_22");
END_REGION

REGION Network 5: 23 - VALVULA 2 VIAS
   "IDB_23"(inConfirmacao_Contator_Lado1 := "IDB_23".outAciona_Lado1,   // "Atuador_Linear_Bifurcada"
            inConfirmacao_Contator_Lado2 := "IDB_23".outAciona_Lado2,
            inSensor_Lado1 := "SENSOR_23_POSICAO_1" OR "teste411",
            inSensor_Lado2 := "SENSOR_23_POSICAO_2" OR "teste412",
            inTempo_Falha := T#20s,
            inEmergencia := "Emergencia_Painel_1",
            inLibera := true,
            Command := "DB_Controle_Equip"."23",
            outAciona_Lado1 => "LIGA_23_SENTIDO_1",
            outAciona_Lado2 => "LIGA_23_SENTIDO_2");
END_REGION

REGION Network 6: 26 - DOSADOR OSCILANTE SILO 1
   "Read_Analogic_Wago"(inValue := "POSICAO_ATUAL_26_SILO1",
                        inValueMax := 100.0,
                        outError => "IDB_26_SILO1".inFalha_Leitura_Posicao,
                        outValue => "IDB_26_SILO1".inPosicao_Atual,
                        ENO => #_w1);
   IF #_w1 THEN
       "IDB_26_SILO1"(inConfirmacao_Contator_Lado1 := "IDB_26_SILO1".outAciona_Lado1,   // "Atuador_Linear_Analogico"
                      inConfirmacao_Contator_Lado2 := "IDB_26_SILO1".outAciona_Lado2,
                      inTolerancia_Erro_Posicao := 5.0,
                      inPosicao_Solicitada_Automatico := "IDB_Controle_Automatico".outPosicao_Atuador_Silo_1,
                      inTempo_Falha := T#20s,
                      inEmergencia := "Emergencia_Painel_1",
                      inLibera := "teste333" <= "DB_Configuracoes".Maquinas.Maximo_Balanca,
                      Command := "DB_Controle_Equip"."26_Silo1",
                      outAciona_Lado1 => "LIGA_26_SILO1_SENTIDO_1",
                      outAciona_Lado2 => "LIGA_26_SILO1_SENTIDO_2");
   END_IF;
END_REGION

REGION Network 7: 26 - DOSADOR OSCILANTE SILO 2
   "Read_Analogic_Wago"(inValue := "POSICAO_ATUAL_26_SILO2",
                        inValueMax := 100.0,
                        outError => "IDB_26_SILO2".inFalha_Leitura_Posicao,
                        outValue => "IDB_26_SILO2".inPosicao_Atual,
                        ENO => #_w1);
   IF #_w1 THEN
       "IDB_26_SILO2"(inConfirmacao_Contator_Lado1 := "IDB_26_SILO2".outAciona_Lado1,   // "Atuador_Linear_Analogico"
                      inConfirmacao_Contator_Lado2 := "IDB_26_SILO2".outAciona_Lado2,
                      inTolerancia_Erro_Posicao := 5.0,
                      inPosicao_Solicitada_Automatico := "IDB_Controle_Automatico".outPosicao_Atuador_Silo_2,
                      inTempo_Falha := T#20s,
                      inEmergencia := "Emergencia_Painel_1",
                      inLibera := "teste333" <= "DB_Configuracoes".Maquinas.Maximo_Balanca,
                      Command := "DB_Controle_Equip"."26_Silo2",
                      outAciona_Lado1 => "LIGA_26_SILO2_SENTIDO_1",
                      outAciona_Lado2 => "LIGA_26_SILO2_SENTIDO_2");
   END_IF;
END_REGION

REGION Network 8: 29 - ROSCA EXTRATORA DA BALANCA
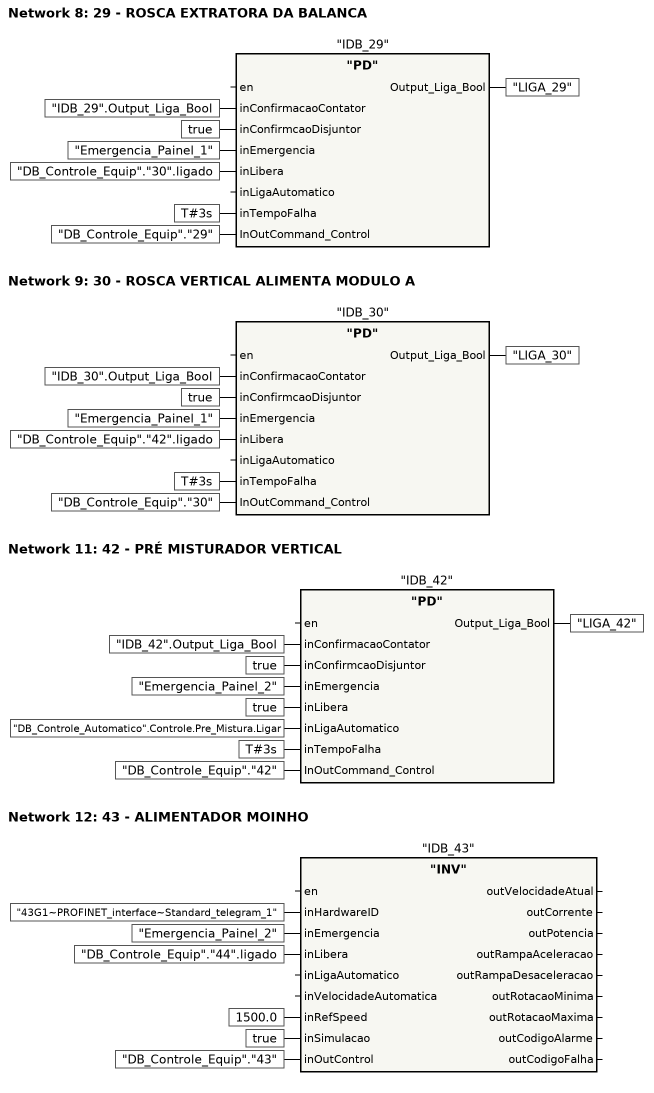
   "IDB_29"(inConfirmacaoContator := "IDB_29".Output_Liga_Bool,   // "PD"
            inConfirmcaoDisjuntor := true,
            inEmergencia := "Emergencia_Painel_1",
            inLibera := "DB_Controle_Equip"."30".ligado,
            inTempoFalha := T#3s,
            InOutCommand_Control := "DB_Controle_Equip"."29",
            Output_Liga_Bool => "LIGA_29");
END_REGION

REGION Network 9: 30 - ROSCA VERTICAL ALIMENTA MODULO A
   "IDB_30"(inConfirmacaoContator := "IDB_30".Output_Liga_Bool,   // "PD"
            inConfirmcaoDisjuntor := true,
            inEmergencia := "Emergencia_Painel_1",
            inLibera := "DB_Controle_Equip"."42".ligado,
            inTempoFalha := T#3s,
            InOutCommand_Control := "DB_Controle_Equip"."30",
            Output_Liga_Bool => "LIGA_30");
END_REGION

REGION Network 10: PAINEL 2 ================================================================
END_REGION

REGION Network 11: 42 - PRÉ MISTURADOR VERTICAL
   "IDB_42"(inConfirmacaoContator := "IDB_42".Output_Liga_Bool,   // "PD"
            inConfirmcaoDisjuntor := true,
            inEmergencia := "Emergencia_Painel_2",
            inLibera := true,
            inLigaAutomatico := "DB_Controle_Automatico".Controle.Pre_Mistura.Ligar,
            inTempoFalha := T#3s,
            InOutCommand_Control := "DB_Controle_Equip"."42",
            Output_Liga_Bool => "LIGA_42");
END_REGION

REGION Network 12: 43 - ALIMENTADOR MOINHO
   "IDB_43"(inHardwareID := "43G1~PROFINET_interface~Standard_telegram_1",   // "INV"
            inEmergencia := "Emergencia_Painel_2",
            inLibera := "DB_Controle_Equip"."44".ligado,
            inRefSpeed := 1500.0,
            inSimulacao := true,
            inOutControl := "DB_Controle_Equip"."43");
END_REGION

REGION Network 13: 44 - MOINHO MARTELO
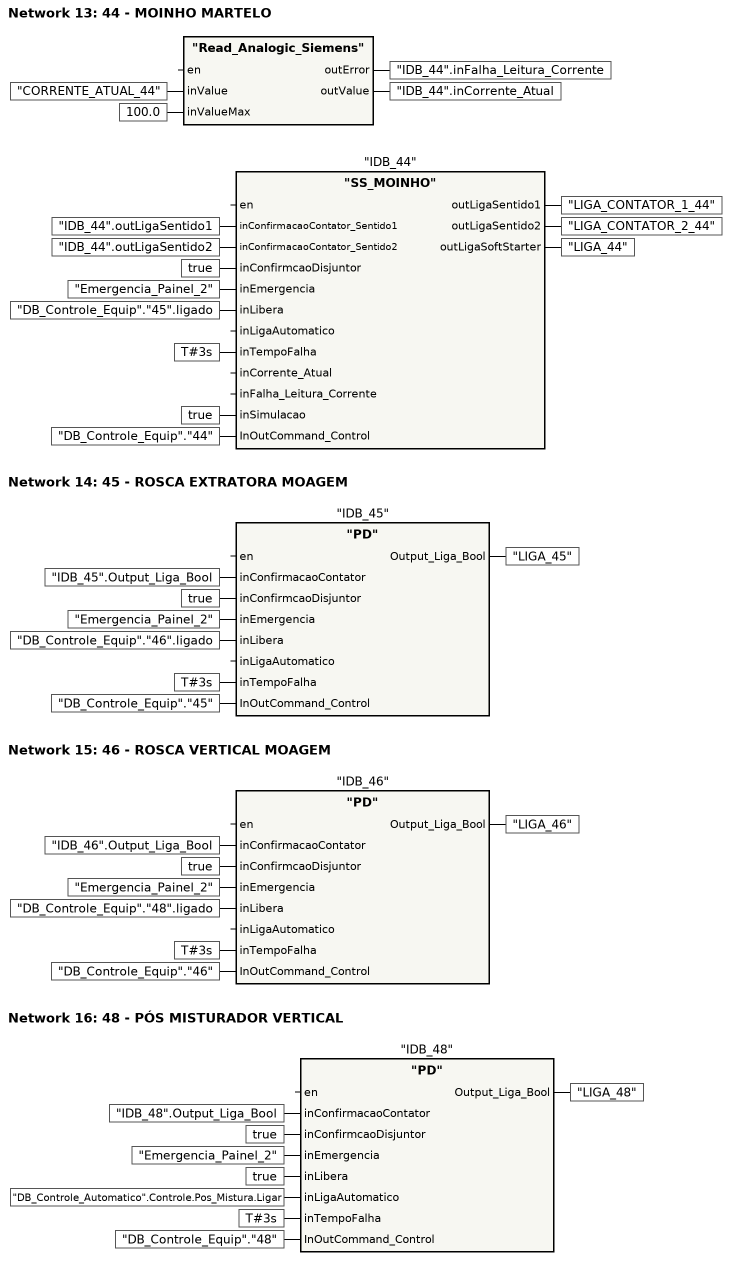
   "Read_Analogic_Siemens"(inValue := "CORRENTE_ATUAL_44",
                           inValueMax := 100.0,
                           outError => "IDB_44".inFalha_Leitura_Corrente,
                           outValue => "IDB_44".inCorrente_Atual);
   "IDB_44"(inConfirmacaoContator_Sentido1 := "IDB_44".outLigaSentido1,   // "SS_MOINHO"
            inConfirmacaoContator_Sentido2 := "IDB_44".outLigaSentido2,
            inConfirmcaoDisjuntor := true,
            inEmergencia := "Emergencia_Painel_2",
            inLibera := "DB_Controle_Equip"."45".ligado,
            inTempoFalha := T#3s,
            inSimulacao := true,
            InOutCommand_Control := "DB_Controle_Equip"."44",
            outLigaSentido1 => "LIGA_CONTATOR_1_44",
            outLigaSentido2 => "LIGA_CONTATOR_2_44",
            outLigaSoftStarter => "LIGA_44");
END_REGION

REGION Network 14: 45 - ROSCA EXTRATORA MOAGEM
   "IDB_45"(inConfirmacaoContator := "IDB_45".Output_Liga_Bool,   // "PD"
            inConfirmcaoDisjuntor := true,
            inEmergencia := "Emergencia_Painel_2",
            inLibera := "DB_Controle_Equip"."46".ligado,
            inTempoFalha := T#3s,
            InOutCommand_Control := "DB_Controle_Equip"."45",
            Output_Liga_Bool => "LIGA_45");
END_REGION

REGION Network 15: 46 - ROSCA VERTICAL MOAGEM
   "IDB_46"(inConfirmacaoContator := "IDB_46".Output_Liga_Bool,   // "PD"
            inConfirmcaoDisjuntor := true,
            inEmergencia := "Emergencia_Painel_2",
            inLibera := "DB_Controle_Equip"."48".ligado,
            inTempoFalha := T#3s,
            InOutCommand_Control := "DB_Controle_Equip"."46",
            Output_Liga_Bool => "LIGA_46");
END_REGION

REGION Network 16: 48 - PÓS MISTURADOR VERTICAL
   "IDB_48"(inConfirmacaoContator := "IDB_48".Output_Liga_Bool,   // "PD"
            inConfirmcaoDisjuntor := true,
            inEmergencia := "Emergencia_Painel_2",
            inLibera := true,
            inLigaAutomatico := "DB_Controle_Automatico".Controle.Pos_Mistura.Ligar,
            inTempoFalha := T#3s,
            InOutCommand_Control := "DB_Controle_Equip"."48",
            Output_Liga_Bool => "LIGA_48");
END_REGION

REGION Network 17: 49 - REGISTRO SAÍDA PÓS MISTURADOR
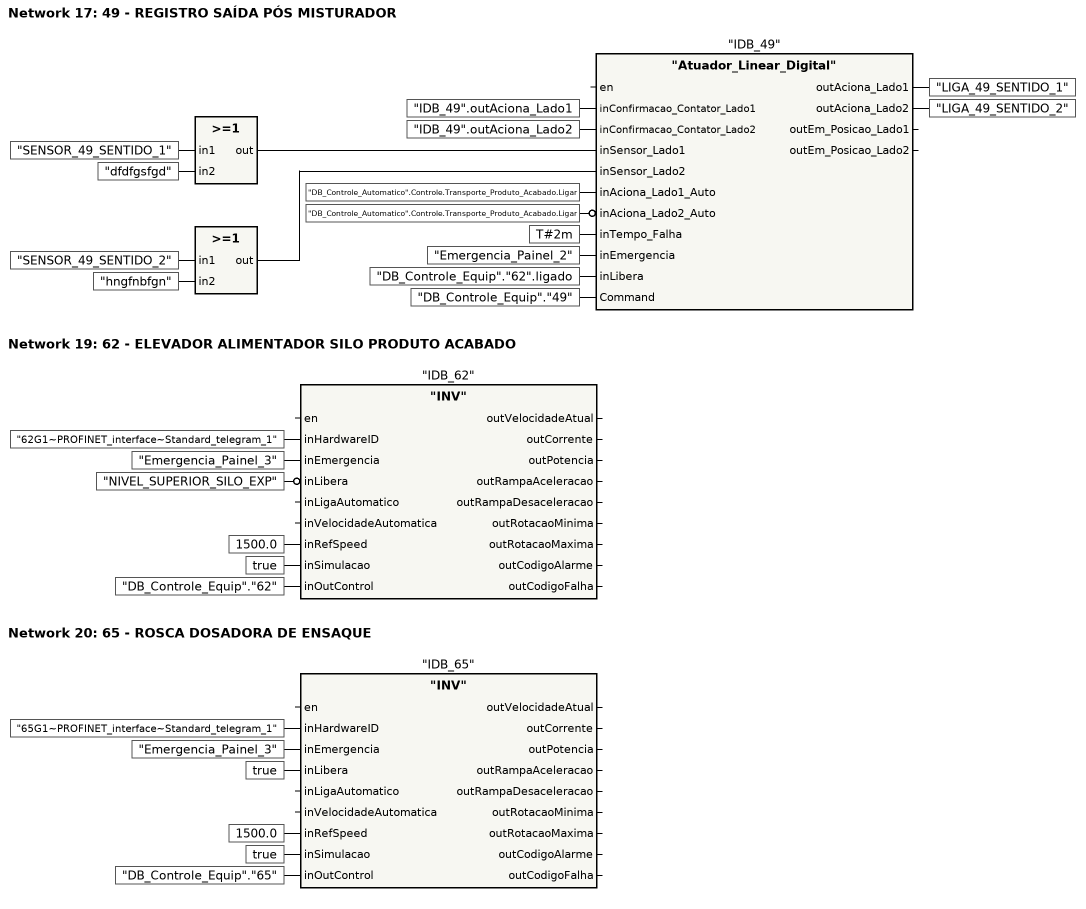
   "IDB_49"(inConfirmacao_Contator_Lado1 := "IDB_49".outAciona_Lado1,   // "Atuador_Linear_Digital"
            inConfirmacao_Contator_Lado2 := "IDB_49".outAciona_Lado2,
            inSensor_Lado1 := "SENSOR_49_SENTIDO_1" OR "dfdfgsfgd",
            inSensor_Lado2 := "SENSOR_49_SENTIDO_2" OR "hngfnbfgn",
            inAciona_Lado1_Auto := "DB_Controle_Automatico".Controle.Transporte_Produto_Acabado.Ligar,
            inAciona_Lado2_Auto := NOT "DB_Controle_Automatico".Controle.Transporte_Produto_Acabado.Ligar,
            inTempo_Falha := T#2m,
            inEmergencia := "Emergencia_Painel_2",
            inLibera := "DB_Controle_Equip"."62".ligado,
            Command := "DB_Controle_Equip"."49",
            outAciona_Lado1 => "LIGA_49_SENTIDO_1",
            outAciona_Lado2 => "LIGA_49_SENTIDO_2");
END_REGION

REGION Network 18: PAINEL 3 ================================================================
END_REGION

REGION Network 19: 62 - ELEVADOR ALIMENTADOR SILO PRODUTO ACABADO
   "IDB_62"(inHardwareID := "62G1~PROFINET_interface~Standard_telegram_1",   // "INV"
            inEmergencia := "Emergencia_Painel_3",
            inLibera := NOT "NIVEL_SUPERIOR_SILO_EXP",
            inRefSpeed := 1500.0,
            inSimulacao := true,
            inOutControl := "DB_Controle_Equip"."62");
END_REGION

REGION Network 20: 65 - ROSCA DOSADORA DE ENSAQUE
   "IDB_65"(inHardwareID := "65G1~PROFINET_interface~Standard_telegram_1",   // "INV"
            inEmergencia := "Emergencia_Painel_3",
            inLibera := true,
            inRefSpeed := 1500.0,
            inSimulacao := true,
            inOutControl := "DB_Controle_Equip"."65");
END_REGION
END_FUNCTION

FUNCTION "FC_Set_Automatico_Equips" : Void   // FC4, FBD
{ S7_Optimized_Access := 'TRUE' }
VERSION : 0.1
BEGIN

REGION Network 1: Jump
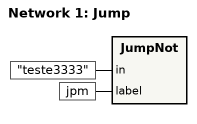
   // no SCL statement known for JumpNot: written as a call
   JumpNot(in := "teste3333", label := jpm);
END_REGION

REGION Network 2: SET Modo Automático em todos os equipamentos
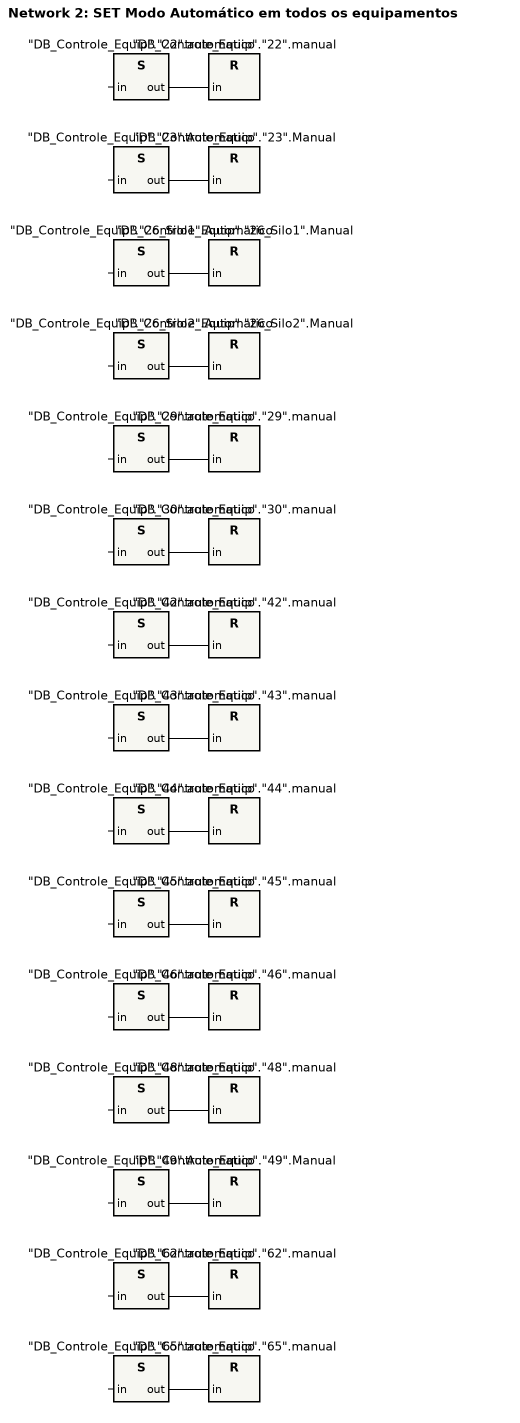
   "DB_Controle_Equip"."22".automatico := TRUE;
   "DB_Controle_Equip"."22".manual := FALSE;
   "DB_Controle_Equip"."23".Automatico := TRUE;
   "DB_Controle_Equip"."23".Manual := FALSE;
   "DB_Controle_Equip"."26_Silo1".Automatico := TRUE;
   "DB_Controle_Equip"."26_Silo1".Manual := FALSE;
   "DB_Controle_Equip"."26_Silo2".Automatico := TRUE;
   "DB_Controle_Equip"."26_Silo2".Manual := FALSE;
   "DB_Controle_Equip"."29".automatico := TRUE;
   "DB_Controle_Equip"."29".manual := FALSE;
   "DB_Controle_Equip"."30".automatico := TRUE;
   "DB_Controle_Equip"."30".manual := FALSE;
   "DB_Controle_Equip"."42".automatico := TRUE;
   "DB_Controle_Equip"."42".manual := FALSE;
   "DB_Controle_Equip"."43".automatico := TRUE;
   "DB_Controle_Equip"."43".manual := FALSE;
   "DB_Controle_Equip"."44".automatico := TRUE;
   "DB_Controle_Equip"."44".manual := FALSE;
   "DB_Controle_Equip"."45".automatico := TRUE;
   "DB_Controle_Equip"."45".manual := FALSE;
   "DB_Controle_Equip"."46".automatico := TRUE;
   "DB_Controle_Equip"."46".manual := FALSE;
   "DB_Controle_Equip"."48".automatico := TRUE;
   "DB_Controle_Equip"."48".manual := FALSE;
   "DB_Controle_Equip"."49".Automatico := TRUE;
   "DB_Controle_Equip"."49".Manual := FALSE;
   "DB_Controle_Equip"."62".automatico := TRUE;
   "DB_Controle_Equip"."62".manual := FALSE;
   "DB_Controle_Equip"."65".automatico := TRUE;
   "DB_Controle_Equip"."65".manual := FALSE;
END_REGION

REGION Network 3: Verifica se todos os equipamentos foram para automatico e reseta a solicitação
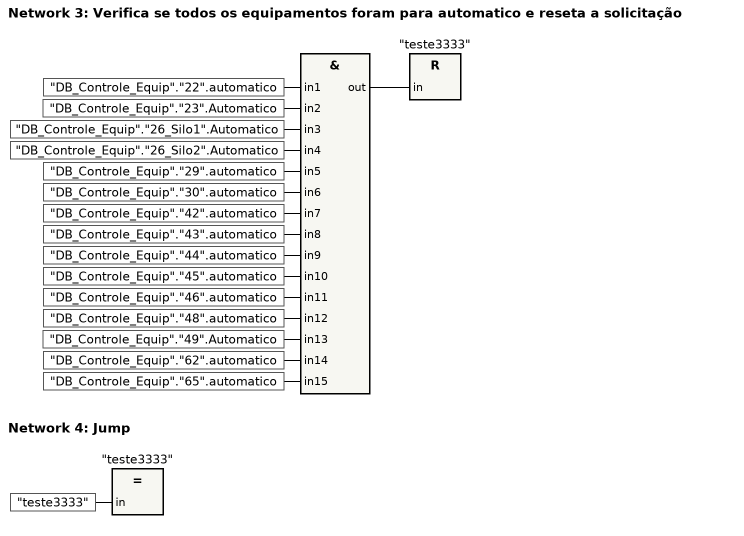
   IF "DB_Controle_Equip"."22".automatico AND "DB_Controle_Equip"."23".Automatico AND "DB_Controle_Equip"."26_Silo1".Automatico AND "DB_Controle_Equip"."26_Silo2".Automatico AND "DB_Controle_Equip"."29".automatico AND "DB_Controle_Equip"."30".automatico AND "DB_Controle_Equip"."42".automatico AND "DB_Controle_Equip"."43".automatico AND "DB_Controle_Equip"."44".automatico AND "DB_Controle_Equip"."45".automatico AND "DB_Controle_Equip"."46".automatico AND "DB_Controle_Equip"."48".automatico AND "DB_Controle_Equip"."49".Automatico AND "DB_Controle_Equip"."62".automatico AND "DB_Controle_Equip"."65".automatico THEN
       "teste3333" := FALSE;
   END_IF;
END_REGION

REGION Network 4: Jump
   jpm:
   "teste3333" := "teste3333";
END_REGION
END_FUNCTION

// folder: FB/Auxiliares

FUNCTION_BLOCK "Liga_Desl_Sequencia"   // FB8, FBD
{ S7_Optimized_Access := 'TRUE' }
VERSION : 0.1
   VAR_INPUT
      inLiga : Bool;
      inQtdMotores : Int;   // Quantos motores serão utilizados de 1 a 10
      inMotor1 : Bool;
      inMotor2 : Bool;
      inMotor3 : Bool;
      inMotor4 : Bool;
      inMotor5 : Bool;
      inMotor6 : Bool;
      inMotor7 : Bool;
      inMotor8 : Bool;
      inMotor9 : Bool;
      inMotor10 : Bool;
   END_VAR
   VAR_OUTPUT
      outMotor1 : Bool;
      outMotor2 : Bool;
      outMotor3 : Bool;
      outMotor4 : Bool;
      outMotor5 : Bool;
      outMotor6 : Bool;
      outMotor7 : Bool;
      outMotor8 : Bool;
      outMotor9 : Bool;
      outMotor10 : Bool;
   END_VAR
   VAR_TEMP   // added for the SCL form of the ladder/FBD networks
      _w1 : Bool;
   END_VAR
BEGIN

REGION Network 1: Liga
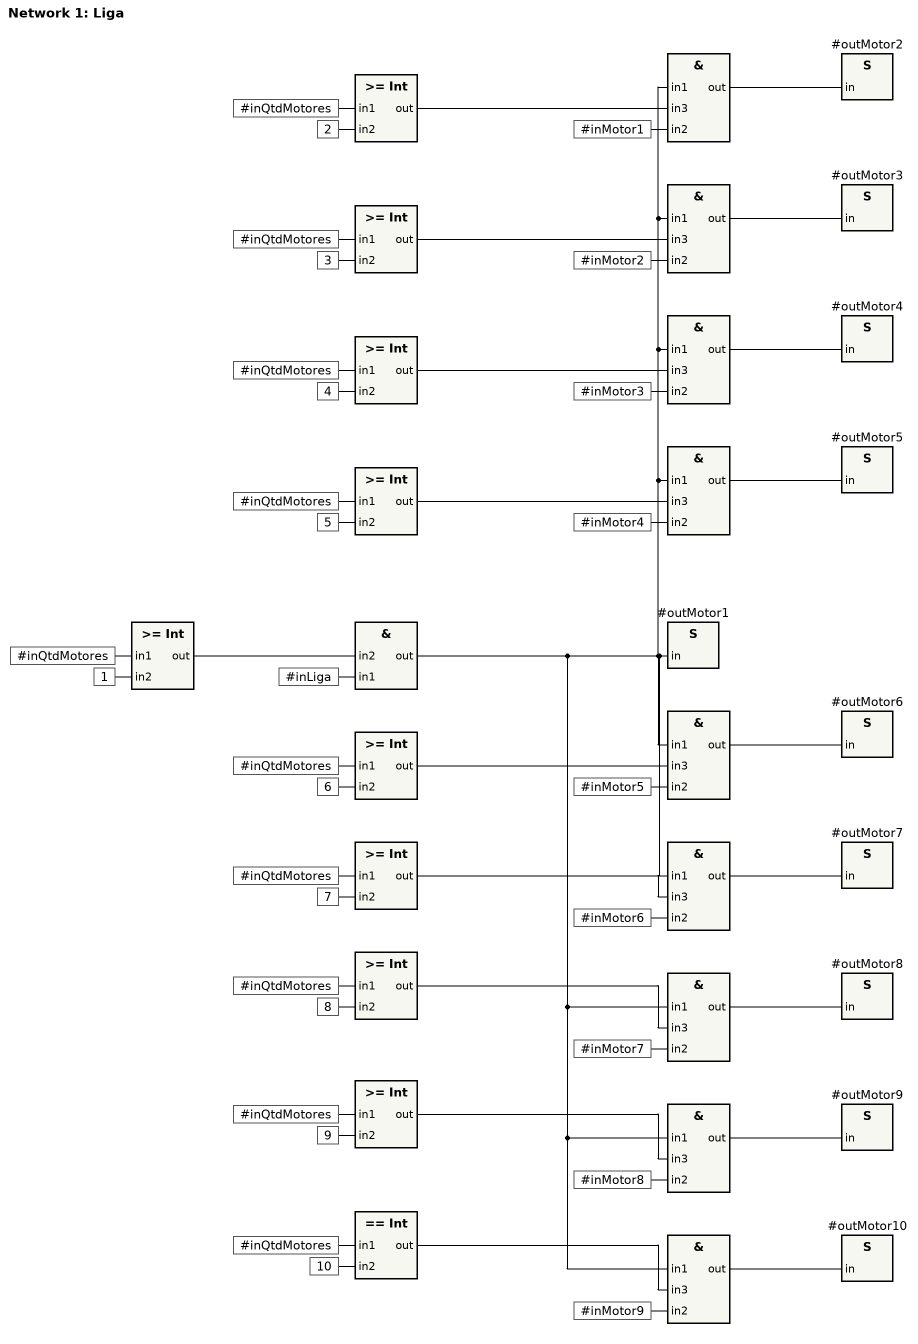
   #_w1 := (#inQtdMotores >= 1) AND #inLiga;
   IF #_w1 THEN #outMotor1 := TRUE; END_IF;
   IF #_w1 AND (#inQtdMotores >= 2) AND #inMotor1 THEN #outMotor2 := TRUE; END_IF;
   IF #_w1 AND (#inQtdMotores >= 3) AND #inMotor2 THEN #outMotor3 := TRUE; END_IF;
   IF #_w1 AND (#inQtdMotores >= 4) AND #inMotor3 THEN #outMotor4 := TRUE; END_IF;
   IF #_w1 AND (#inQtdMotores >= 5) AND #inMotor4 THEN #outMotor5 := TRUE; END_IF;
   IF #_w1 AND (#inQtdMotores >= 6) AND #inMotor5 THEN #outMotor6 := TRUE; END_IF;
   IF #_w1 AND (#inQtdMotores >= 7) AND #inMotor6 THEN #outMotor7 := TRUE; END_IF;
   IF #_w1 AND (#inQtdMotores >= 8) AND #inMotor7 THEN #outMotor8 := TRUE; END_IF;
   IF #_w1 AND (#inQtdMotores >= 9) AND #inMotor8 THEN #outMotor9 := TRUE; END_IF;
   IF #_w1 AND (#inQtdMotores = 10) AND #inMotor9 THEN #outMotor10 := TRUE; END_IF;
END_REGION

REGION Network 2: Desliga
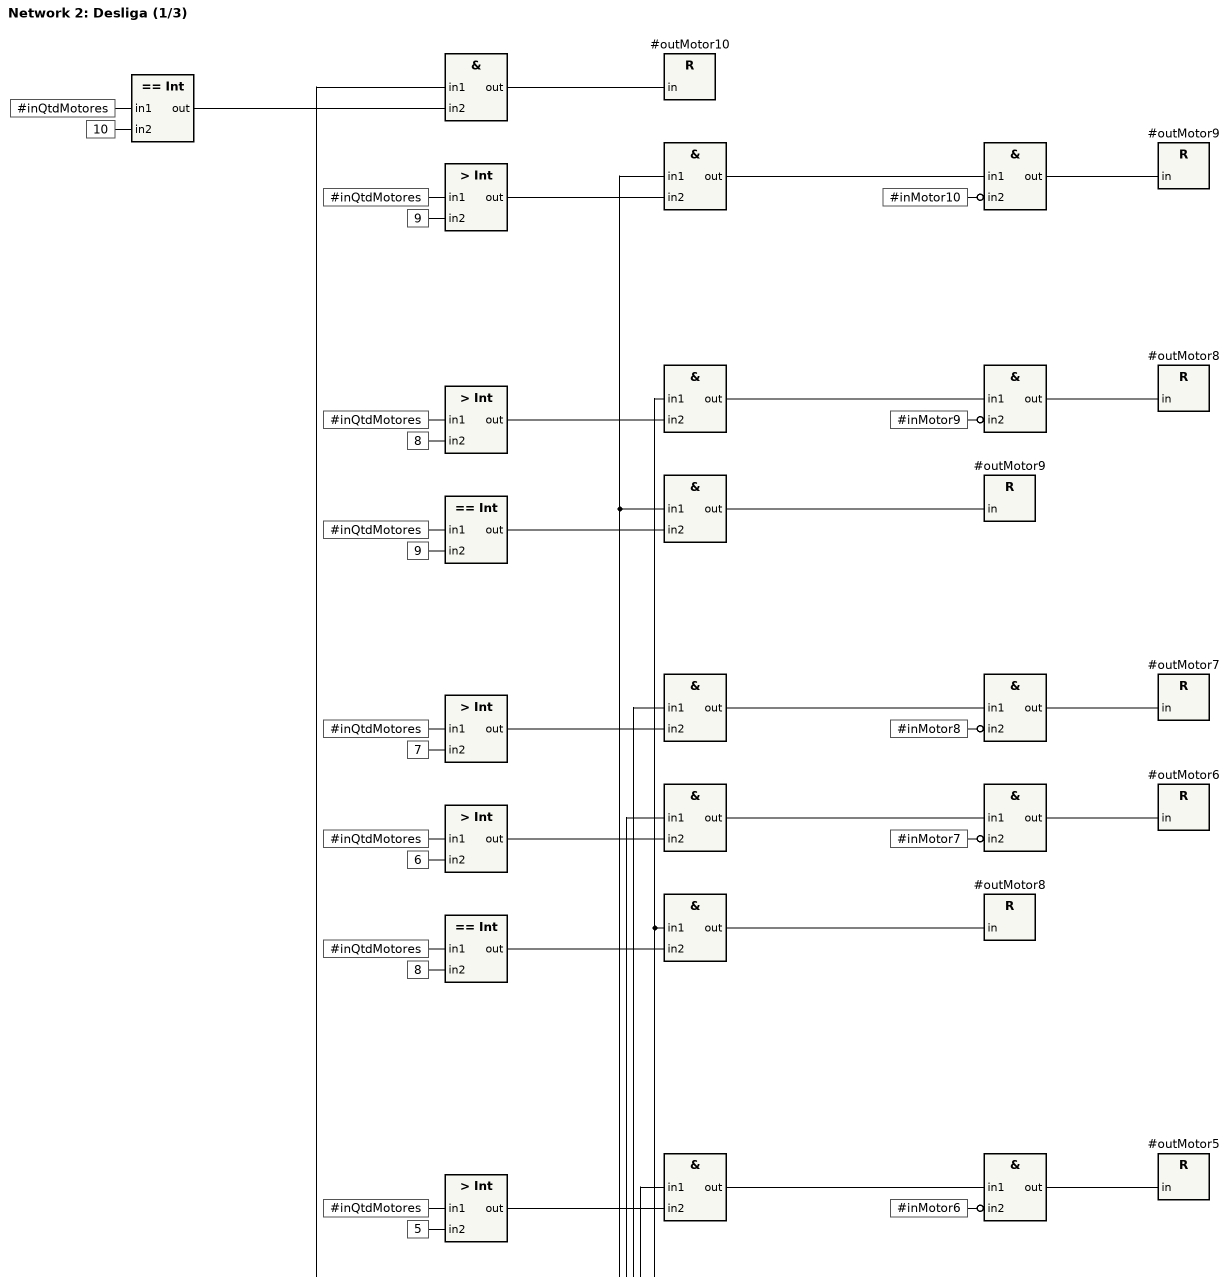
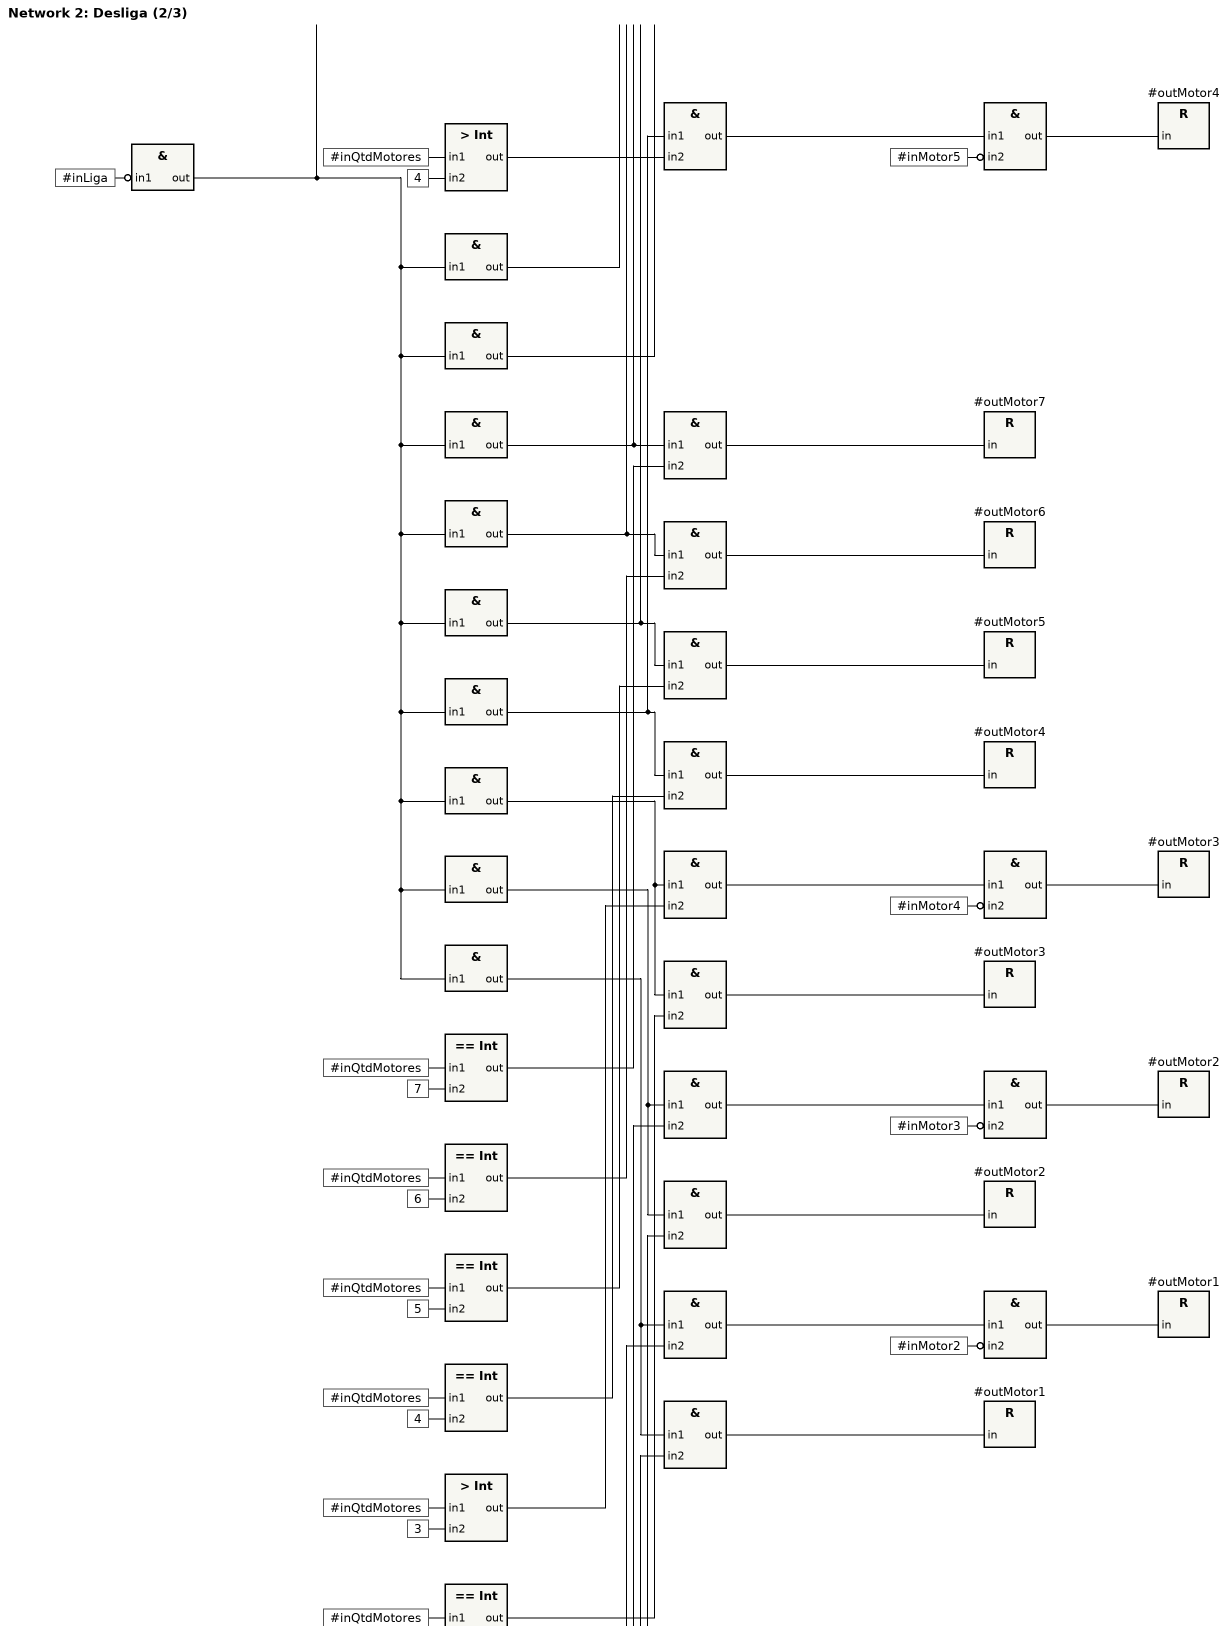
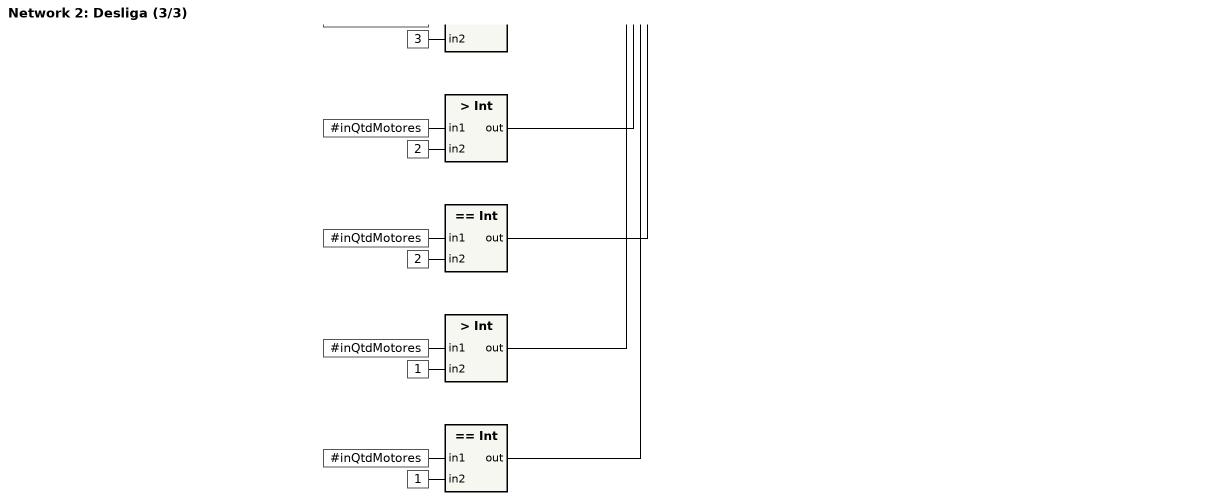
   IF NOT #inLiga AND (#inQtdMotores = 10) THEN #outMotor10 := FALSE; END_IF;
   IF NOT #inLiga AND (#inQtdMotores > 9) AND NOT #inMotor10 THEN #outMotor9 := FALSE; END_IF;
   IF NOT #inLiga AND (#inQtdMotores = 9) THEN #outMotor9 := FALSE; END_IF;
   IF NOT #inLiga AND (#inQtdMotores > 8) AND NOT #inMotor9 THEN #outMotor8 := FALSE; END_IF;
   IF NOT #inLiga AND (#inQtdMotores = 8) THEN #outMotor8 := FALSE; END_IF;
   IF NOT #inLiga AND (#inQtdMotores > 7) AND NOT #inMotor8 THEN #outMotor7 := FALSE; END_IF;
   IF NOT #inLiga AND (#inQtdMotores = 7) THEN #outMotor7 := FALSE; END_IF;
   IF NOT #inLiga AND (#inQtdMotores > 6) AND NOT #inMotor7 THEN #outMotor6 := FALSE; END_IF;
   IF NOT #inLiga AND (#inQtdMotores = 6) THEN #outMotor6 := FALSE; END_IF;
   IF NOT #inLiga AND (#inQtdMotores > 5) AND NOT #inMotor6 THEN #outMotor5 := FALSE; END_IF;
   IF NOT #inLiga AND (#inQtdMotores = 5) THEN #outMotor5 := FALSE; END_IF;
   IF NOT #inLiga AND (#inQtdMotores > 4) AND NOT #inMotor5 THEN #outMotor4 := FALSE; END_IF;
   IF NOT #inLiga AND (#inQtdMotores = 4) THEN #outMotor4 := FALSE; END_IF;
   IF NOT #inLiga AND (#inQtdMotores > 3) AND NOT #inMotor4 THEN #outMotor3 := FALSE; END_IF;
   IF NOT #inLiga AND (#inQtdMotores = 3) THEN #outMotor3 := FALSE; END_IF;
   IF NOT #inLiga AND (#inQtdMotores > 2) AND NOT #inMotor3 THEN #outMotor2 := FALSE; END_IF;
   IF NOT #inLiga AND (#inQtdMotores = 2) THEN #outMotor2 := FALSE; END_IF;
   IF NOT #inLiga AND (#inQtdMotores > 1) AND NOT #inMotor2 THEN #outMotor1 := FALSE; END_IF;
   IF NOT #inLiga AND (#inQtdMotores = 1) THEN #outMotor1 := FALSE; END_IF;
END_REGION
END_FUNCTION_BLOCK

FUNCTION_BLOCK "Horimetro_REV01"   // FB13, FBD
{ S7_Optimized_Access := 'TRUE' }
VERSION : 0.1
   VAR_INPUT
      Input_Liga_Horimetro_Bool : Bool;
      Input_SP_Manutencao : DInt;
   END_VAR
   VAR_OUTPUT
      Output_Hora_Parcial_DInt : DInt;
      Output_Hora_Total_DInt : DInt;
      Output_ManutencaoRequeirda : Bool;
   END_VAR
   VAR_IN_OUT
      InOut_Reset_Parcial_Bool : Bool;
      InOut_Reset_Total_Bool : Bool;
   END_VAR
   VAR
      Static_TONR_Parcial : TONR_TIME;
   END_VAR
   VAR RETAIN
      Static_Contador_Horas_Parcial : CTU_DINT;
   END_VAR
   VAR
      Static_TONR_Total : TONR_TIME;
   END_VAR
   VAR RETAIN
      Static_Contador_Horas_Total : CTU_DINT;
   END_VAR
   VAR
      Static_Reset_Parcial : Bool;
      Static_Reset_Total : Bool;
   END_VAR
BEGIN

REGION Network 1: Horimetro Parcial
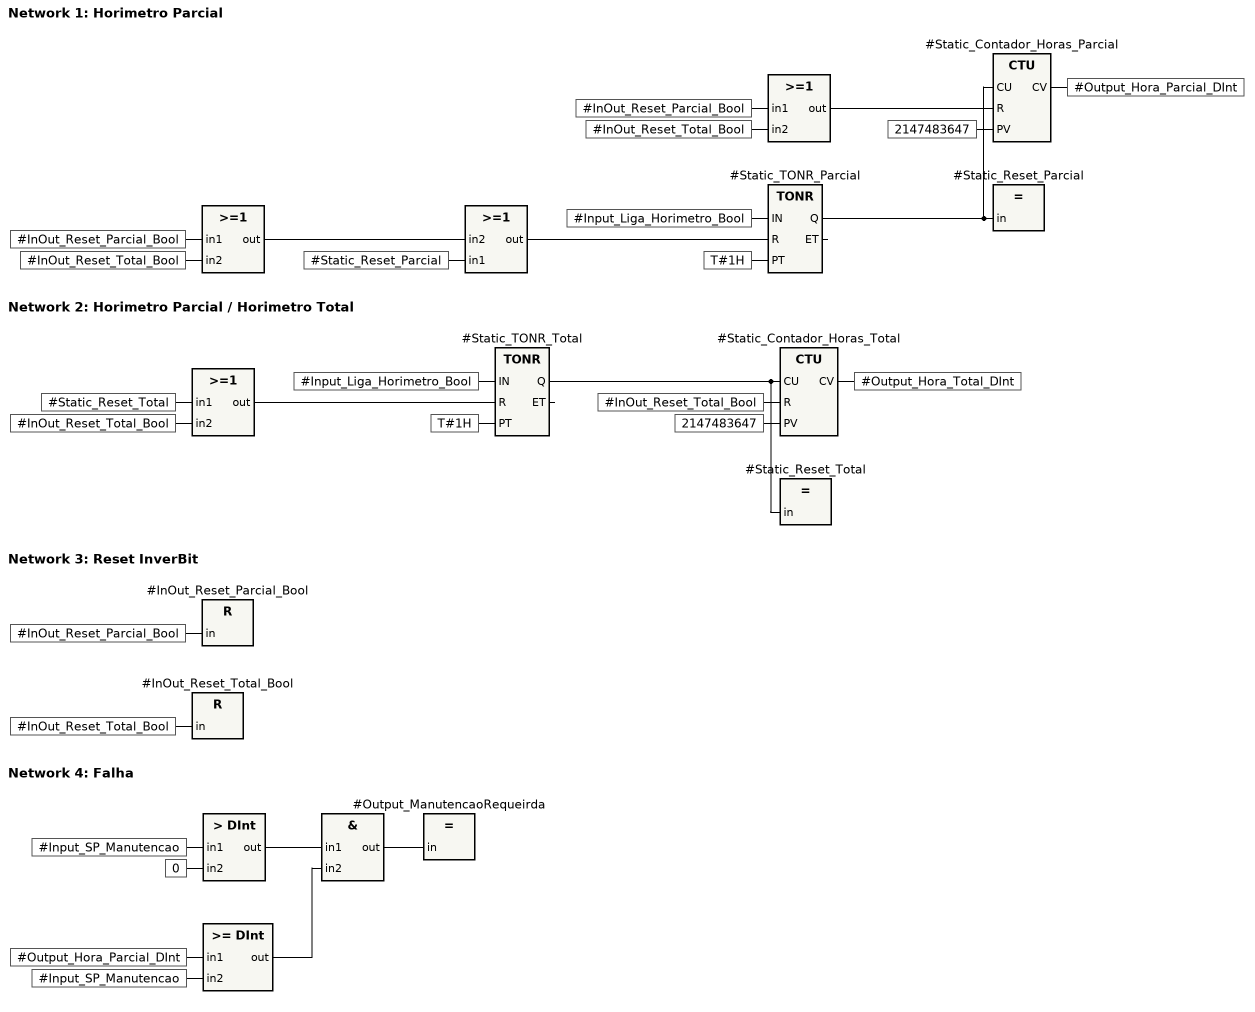
   #Static_TONR_Parcial(IN := #Input_Liga_Horimetro_Bool,   // TONR
                        R := #InOut_Reset_Parcial_Bool OR #InOut_Reset_Total_Bool OR #Static_Reset_Parcial,
                        PT := T#1H);
   #Static_Contador_Horas_Parcial(CU := #Static_TONR_Parcial.Q,   // CTU
                           R := #InOut_Reset_Parcial_Bool OR #InOut_Reset_Total_Bool,
                           PV := 2147483647,
                           CV => #Output_Hora_Parcial_DInt);
   #Static_Reset_Parcial := #Static_TONR_Parcial.Q;
END_REGION

REGION Network 2: Horimetro Parcial / Horimetro Total
   #Static_TONR_Total(IN := #Input_Liga_Horimetro_Bool,   // TONR
                      R := #Static_Reset_Total OR #InOut_Reset_Total_Bool,
                      PT := T#1H);
   #Static_Contador_Horas_Total(CU := #Static_TONR_Total.Q,   // CTU
                           R := #InOut_Reset_Total_Bool,
                           PV := 2147483647,
                           CV => #Output_Hora_Total_DInt);
   #Static_Reset_Total := #Static_TONR_Total.Q;
END_REGION

REGION Network 3: Reset InverBit
   IF #InOut_Reset_Parcial_Bool THEN #InOut_Reset_Parcial_Bool := FALSE; END_IF;
   IF #InOut_Reset_Total_Bool THEN #InOut_Reset_Total_Bool := FALSE; END_IF;
END_REGION

REGION Network 4: Falha
   #Output_ManutencaoRequeirda := (#Input_SP_Manutencao > 0) AND (#Output_Hora_Parcial_DInt >= #Input_SP_Manutencao);
END_REGION
END_FUNCTION_BLOCK

FUNCTION_BLOCK "SINA_SPEED"   // FB285, SCL
TITLE = 'Speed Control with SINAMICS and S7'
{ S7_Optimized_Access := 'TRUE' }
AUTHOR : DRVDPS7
FAMILY : DRIVES
NAME : SINA_SPD
VERSION : 5.0
// Copyright (C) Siemens AG 2012. All Rights Reserved. Confidential
// -------------------------------------------------------------------------------------- 
// SINA_SPEED: Drehzahlregelung mit dem Antriebsbaustein SINAMICS S120/G120 <-> S7-1200
// ------------------------------------------------------------------------------------- Ersteller: Siemens AG Erlangen A&D MC PM   Datum:  07.07.10        Vers.:2.1
// Ã„nderung:  J.B. Typical Team                       07.12.12              2.2
//     Umsetzung in SCL / TIA 
// Ã„nderung:  J.B. Typical Team                       29.04.13              2.3
//     1. "Q" an den AusgÃ¤nge entfernen
//     2. Neuer Ausgang PwrInhibit
// Ã„nderung:  J.B. Typical Team                       28.06.13              2.4
//     Ã„nderung HW-Zugriff Ã¼ber LOG2MOD
//      
// Ã„nderung:  J.B. Typical Team                       18.07.13              2.5
//     Ã„nderung HW-Zugriff Ã¼ber zwei HW-EingÃ¤nge
// 
// Ã„nderung:  J.B. Typical Team                       17.07.14              3.0
//     Optimmierung
// 
// Ã„nderung:  J.B. Typical Team                       30.07.14              4.0
//     Festlegung auf einheitlicher neuer Version 4.0
// 
// Ã„nderung:  P.Z. Typical Team                       03.12.15              4.1
//     Schnittstelle an Programmierleitfadeb TIA-Potal angepasst
//     zusÃ¤tzlicher Eingang "ConfigAxis" fÃ¼r STW-Bits
// 
// Ã„nderung:  G.F. Typical Team                       01.03.16              4.2
//     Sollwert auf INT - Grenzen begrenzt
// Ã„nderung:  F.G. Typical Team                       13.09.16              4.3
//     Ausgabewerte am Ausgang "Status" angepasst 
// 
// Ã„nderung:  G.F. Typical Team                       11.01.17              5.0
//     - Festlegung auf einheitlicher neuer Version 5.0 
// 
// Bibliothek V7
// Funktion: Drehzahlregelung mit dem Antriebsbaustein SINAMICS S120/G120 <-> S7-1200
// ********************************************************************************************************************************************************
// ************************************************************************FB283***************************************************************************
// ********************************************************************************************************************************************************
   VAR_INPUT
      EnableAxis : Bool := 0;   // 0-->1; 1 = Enable the drive (OFF2 / OFF 3 are 1 in default status) (OFF1 = 0-->1) / 0-->1 = Einschalten des Antriebs (OFF1 = 0-->1)
      AckError : Bool := 0;   // 1 = Acknowledge drive error / 1 = Fehlerquitierung angestoßen
      SpeedSp : Real := 0.0;   // Speed standardises with the standardisation factor / Drehzahlsollwert [rpm]
      RefSpeed : Real := 0.0;   // Standardisation factor of speed / Referenzdrehzahl (p2000 in [rpm])
      ConfigAxis : Word := 16#003F;   // binary programmed input to control all functions in the telegram without its own function block input / Binärcodierter Eingang zur Ansteuerung aller nicht als Bausteineingang verfügbaren Steuerbits
      HWIDSTW : Hw_Io := 0;   // Hardware Identifer set point slot / Hardware Identifer des Sollwert Slots
      HWIDZSW : Hw_Io := 0;   // Hardware Identifer actual value slot / Hardware Identifer des Istwert Slots
   END_VAR
   VAR_OUTPUT
      AxisEnabled : Bool := 0;   // 1 = Drive is enabled / 1 = Antrieb in Betrieb
      Lockout : Bool := 0;   // 1 = Drive lockout active / 1 = Einschaltsperre aktiv
      ActVelocity : Real := 0.0;   // Actual in [U/min] / Aktuelle Geschwindigkeit [rpm]
      Error : Bool := 0;   // 1 = Error (FB and Infeed) / 1 = Fehler im Baustein / Antrieb
      Status : Word := 0;   // Status output (7002 = FB in operation; 8xxx = error description - read the manual) / Statusausgabe (7002 = FB in Betrieb; 8xxx = Feherbeschreibung siehe Doku)
      DiagId : Word := 16#0000;   // Error codes of the cyclic system funtion blocks DPWR / DPRD_DAT / Fehlercode der zyklischen Systemfunktionen DPWR / DPRD_DAT
   END_VAR
   VAR
      sxSendBuf : Struct   // Send buffer
         STW1 : Word := WORD#16#0000;   // STW1sxSTW1 : STRUCT Bit08 : BOOL:=False; // ST-Wort-1 Bit 08 --> Reserve Bit09 : BOOL:=False; // ST-Wort-1 Bit 09 --> Reserve Bit10 : BOOL:=True; // ST-Wort-1 Bit 10 --> FÃ¼hrung durch PLC Dir : BOOL:=False; // ST-Wort-1 Bit 11 --> Direction Bit12 : BOOL:=False; // ST-Wort-1 Bit 12 --> Haltebremse unbedingt Ã¶ffnen Bit13 : BOOL:=False; // ST-Wort-1 Bit 13 --> Motorpotenziometer Sollwert hÃ¶her Bit14 : BOOL:=False; // ST-Wort-1 Bit 14 --> Motorpotenziometer Sollwert tiefer Bit15 : BOOL:=False; // ST-Wort-1 Bit 15 --> Reserviert Off1 : BOOL:=False; // ST-Wort-1 Bit 00 --> OFF1/ON (flanks acceptance) Off2 : BOOL:=True; // ST-Wort-1 Bit 01 --> OFF2/ON (enable possible) Off3 : BOOL:=True; // ST-Wort-1 Bit 02 --> OFF3/ON (enable possible) InvEn : BOOL:=True; // ST-Wort-1 Bit 03 --> Enable controller RampEn : BOOL:=True; // ST-Wort-1 Bit 04 --> Ramp enable RampOn : BOOL:=True; // ST-Wort-1 Bit 05 --> Ramp On SpEn : BOOL:=True; // ST-Wort-1 Bit 06 --> Speed set point enable AckFlt : BOOL:=False; // ST-Wort-1 Bit 07 --> Acknowledge fault END_STRUCT;
         Velocity : Word := WORD#16#0000;   // Setpoint of velocity
      END_STRUCT;
      sxRecvBuf : Struct   // Receive buffer
         ZSW1 : Word := WORD#16#0000;   // ZSW1sxZSW1 : STRUCT SpDev : BOOL:=False; // ZSW-Wort-1 = Schleppfehler im Toleranzbereich Pcd : BOOL:=False; // ZSW-Wort-1 = PZD-FÃ¼hrung erreicht Comp : BOOL:=False; // ZSW-Wort-1 = Zielposition erreicht CurLim : BOOL:=False; // ZSW-Wort-1 = Referenzpunkt gesetzt Brake : BOOL:=False; // ZSW-Wort-1 = Haltebremse Ã¶ffnen Motover : BOOL:=False; // ZSW-Wort-1 = keine Warnung Ãœbertemperatur Motor Dir : BOOL:=False; // ZSW-Wort-1 = Direction Invover : BOOL:=False; // ZSW-Wort-1 = keine Warnung thermische Ãœberlast Leistungsteil Rts : BOOL:=False; // ZSW-Wort-1 = Ready to power up / to start Rdy : BOOL:=False; // ZSW-Wort-1 = Ready to operate IOp : BOOL:=False; // ZSW-Wort-1 = In operation (operation enabled) Fault : BOOL:=False; // ZSW-Wort-1 = Fault present NoOff2 : BOOL:=False; // ZSW-Wort-1 = OFF2 inactive NoOff3 : BOOL:=False; // ZSW-Wort-1 = OFF3 inactive Inhibit : BOOL:=False; // ZSW-Wort-1 = Power ON inhibit active Alarm : BOOL:=False; // ZSW-Wort-1 = Alarm / Warning present END_STRUCT;
         Velocity : Word := WORD#16#0000;   // Feedback of velocity
      END_STRUCT;
   END_VAR
   VAR_TEMP
      piRetSFC : Int;   // Status for fault analysis
      piCount : Int;   // Freely available counter variable 3
      prVelocity : Real;   // velocity
      pdRecvBuf : DWord;   // Buffer of Recv-Value
      pdSendBuf : DWord;   // Buffer of Send-Value
      phLAddr : Hw_Io;   // Start addr from the I/O process image area of mod (DEC) for DPWR_DAT/DPRD_DAT / Adresse des Sollwert Slots
      swSendBuf : Array[0..1] of Word;   // Sendepuffer
      swRecvBuf : Array[0..1] of Word;   // Empfangspuffer Static variables
   END_VAR
BEGIN

   //=============================================================================
   //SIEMENS AG
   //(c)Copyright 2017 All Rights Reserved
   //-----------------------------------------------------------------------------
   // Library: DriveLib
   // Tested with: S7-1516-3 PN/DP V1.8
   // Engineering: TIA Portal V14
   // Restrictions: -
   // Requirements: S7-1200 / S7-1500
   // Functionality: cyclic communication between a SINAMICS a PLC.
   //                If in HWConfig Std.TLG 1 is projected 2 PZD-words are exchanged
   //                in every bus cycle.
   //                The parametrisation of these words is described in the manual of the
   //                SINAMICS
   //=============================================================================

   // Schreibdaten zusammenstellen
   // Steuerword aufbereiten

   #sxSendBuf.STW1.%X0 := #EnableAxis;
   #sxSendBuf.STW1.%X1 := #ConfigAxis.%X0;
   #sxSendBuf.STW1.%X2 := #ConfigAxis.%X1;
   #sxSendBuf.STW1.%X3 := #ConfigAxis.%X2;
   #sxSendBuf.STW1.%X4 := #ConfigAxis.%X3;
   #sxSendBuf.STW1.%X5 := #ConfigAxis.%X4;
   #sxSendBuf.STW1.%X6 := #ConfigAxis.%X5;
   #sxSendBuf.STW1.%X10 := TRUE;
   #sxSendBuf.STW1.%X11 := #ConfigAxis.%X6;
   #sxSendBuf.STW1.%X7 := #AckError;

   // Geschwindigkeit
   IF #RefSpeed <> 0 THEN
     #prVelocity := #SpeedSp * (16384.0 / #RefSpeed);
     // Limit REAL - Variable to INT - Limits
     IF #prVelocity > 32767 THEN
       #prVelocity := 32767;
     ELSIF #prVelocity < -32768 THEN
       #prVelocity := -32768;
     ELSE
       ; // not needed
     END_IF;
     #sxSendBuf.Velocity := INT_TO_WORD(REAL_TO_INT(#prVelocity));

   ELSE
     #sxSendBuf.Velocity := W#16#0;
   END_IF;
   #swSendBuf[0] := #sxSendBuf.STW1;
   #swSendBuf[1] := #sxSendBuf.Velocity;

   //Prozessdaten zur Signalbaugruppe schreiben
   #piRetSFC := DPWR_DAT(LADDR := #HWIDSTW,
                         RECORD := #swSendBuf);

   // Fehler der RÃ¼ckmeldung ausgeben
   #DiagId := INT_TO_WORD(#piRetSFC);

   //kein Fehler beim Schreiben
   IF #piRetSFC = 0 THEN

     //kein Fehler beim Schreiben
     IF #piRetSFC = 0 THEN

       //Prozessdaten von der Signalbaugruppe lesen
       #piRetSFC := DPRD_DAT(LADDR := #HWIDZSW,
                             RECORD => #swRecvBuf);

       // Fehler der RÃ¼ckmeldung ausgeben
       #DiagId := INT_TO_WORD(#piRetSFC);
     END_IF;

     //Fehler beim Lesen (Profibus-Kommunikation unterbrochen)
     IF #piRetSFC <> 0 THEN

       // Fehler
       #Error := TRUE;
       #Status := 16#8600;

       // Zustandsworte lÃ¶schen
       #sxRecvBuf.ZSW1.%X8 := 0;
       #sxRecvBuf.ZSW1.%X9 := 0;
       #sxRecvBuf.ZSW1.%X10 := 0;
       #sxRecvBuf.ZSW1.%X11 := 0;
       #sxRecvBuf.ZSW1.%X12 := 0;
       #sxRecvBuf.ZSW1.%X13 := 0;
       #sxRecvBuf.ZSW1.%X14 := 0;
       #sxRecvBuf.ZSW1.%X15 := 0;
       #sxRecvBuf.ZSW1.%X0 := 0;
       #sxRecvBuf.ZSW1.%X1 := 0;
       #sxRecvBuf.ZSW1.%X2 := 0;
       #sxRecvBuf.ZSW1.%X3 := 0;
       #sxRecvBuf.ZSW1.%X4 := 0;
       #sxRecvBuf.ZSW1.%X5 := 0;
       #sxRecvBuf.ZSW1.%X6 := 0;
       #sxRecvBuf.ZSW1.%X7 := 0;


       (*#sxRecvBuf.sxZSW1.SpDev   := 0;
       #sxRecvBuf.sxZSW1.Pcd     := 0;
       #sxRecvBuf.sxZSW1.Comp    := 0;
       #sxRecvBuf.sxZSW1.CurLim  := 0;
       #sxRecvBuf.sxZSW1.Brake   := 0;
       #sxRecvBuf.sxZSW1.Motover := 0;
       #sxRecvBuf.sxZSW1.Dir     := 0;
       #sxRecvBuf.sxZSW1.Invover := 0;
       #sxRecvBuf.sxZSW1.Rts     := 0;
       #sxRecvBuf.sxZSW1.Rdy     := 0;
       #sxRecvBuf.sxZSW1.IOp     := 0;
       #sxRecvBuf.sxZSW1.Fault   := 0;
       #sxRecvBuf.sxZSW1.NoOff2  := 0;
       #sxRecvBuf.sxZSW1.NoOff3  := 0;
       #sxRecvBuf.sxZSW1.Inhibit := 0;
       #sxRecvBuf.sxZSW1.Alarm   := 0;*)

       #sxRecvBuf.Velocity := W#16#00;

       // Werte auslesen
     ELSE
       #sxRecvBuf.ZSW1 := #swRecvBuf[0];
       #sxRecvBuf.Velocity := #swRecvBuf[1];

       // ZSW1 aufbereiten                       
       #AxisEnabled := #sxRecvBuf.ZSW1.%X2;
       #Error := #sxRecvBuf.ZSW1.%X3 OR #sxRecvBuf.ZSW1.%X6;
       #Lockout := #sxRecvBuf.ZSW1.%X6;

       // Fehler auswerten
       IF #sxRecvBuf.ZSW1.%X3 THEN
         #Status := 16#8401;
       ELSIF #sxRecvBuf.ZSW1.%X6 THEN
         #Status := 16#8402;
       ELSE
         #Status := 16#7002;
       END_IF;

       (*#Busy       := #sxRecvBuf.sxZSW1.IOp;
       #Error      := #sxRecvBuf.sxZSW1.Fault OR #sxRecvBuf.sxZSW1.Inhibit;
       #PwrInhibit := #sxRecvBuf.sxZSW1.Inhibit;            

       // Fehler auswerten
       IF #sxRecvBuf.sxZSW1.Fault THEN
           #ErrorId := 1;
       ELSIF #sxRecvBuf.sxZSW1.Inhibit THEN 
           #ErrorId := 2;
       ELSE
           #ErrorId := 0;    
       END_IF;*)

       // Geschwindigkeit
       IF #RefSpeed <> 0 THEN
         #ActVelocity := INT_TO_REAL(WORD_TO_INT(#sxRecvBuf.Velocity)) / (16384.0 / #RefSpeed);
       ELSE
         #ActVelocity := 0.0;
       END_IF;
     END_IF;
   ELSE

     // Fehler
     #Error := TRUE;
     #Status := 16#8601;

   END_IF;
END_FUNCTION_BLOCK

FUNCTION_BLOCK "SINA_PARA"   // FB286, SCL
TITLE = 'parameter exchange between SINAMICS and S7'
{ S7_Optimized_Access := 'TRUE' }
AUTHOR : DRVDPS7
FAMILY : DRIVES
NAME : SINA_PAR
VERSION : 5.0
// Copyright (C) Siemens AG 2012. All Rights Reserved. Confidential
// --------------------------------------------------------------------------- 
// SINA_PARA: Austausch 15 beliebiger Parameter zwischen SINAMICS S120/G120 <-> S7
// -------------------------------------------------------------------------- Ersteller: Siemens AG Erlangen A&D MC PM   Datum:  07.07.10        Vers.:2.1
// Änderung:  J.B. Typical Team                       09.01.13              2.2
//     Umsetzung in SCL / TIA 
// Änderung:  J.B. Typical Team                       29.04.13              2.3 
//     "Q" an den Ausgänge entfernen
//      
// Änderung:  J.B. Typical Team                       28.06.13              2.4
//     HW-Zugriffsermittlung über LOG2MOD
// 
// Änderung:  J.B. Typical Team                       25.07.13              2.5
//     Wiederholfaktor bei temporäre Fehler
//         
// Änderung:  J.B. Typical Team                       24.09.13              2.6
//     Konvertierungsfehler
//     
// Änderung:  J.B. Typical Team                       05.10.13              2.7
//     Fehlerkorrektur im Antworttelegramm bei 
//     Änderung
// Änderung:  J.B. Typical Team                       16.12.13              2.8
//     weiterhin Fehlerkorrektur im Antworttelegramm bei 
//     Änderung
//     
// Änderung:  J.B. Typical Team                       15.01.14              2.9
//     weiterhin Fehlerkorrektur im Antworttelegramm bei 
//     Änderung
// Änderung:  J.B. Typical Team                       17.07.14              3.0
//     Nun mit Optimierung 
// 
// Änderung:  J.B. Typical Team                       30.07.14              4.0
//     Festlegung auf einheitlicher neuer Version 4.0
// 
// Änderung:  G.F. Typical Team                       20.05.15              4.1
//     Fehler bei der Umrechnung der Parameterwerte behoben
// 
// Änderung:  G.F. Typical Team                       15.09.15              4.2
//     Defaultwert des Parameters AxisNo von 0 auf 1 geändert
// 
// Änderung:  G.F. Typical Team                       06.10.15              4.3
//     Defaultwert der Parameter AxisNo, ParaNo und Done von 0 auf 1 geändert
//     und Parameter swParaError gezielt auf 0 gesetzt
// 
// Änderung:  J.B. Typical Team                       08.12.15              4.4
//     1. Wenn beim Parameter "Lesen" ein Fehler zurück gemeldet wird, 
//     soll das "Schreiben" abgebrochen werden
// 
//     2. Für den Datentyp DWORD mit/ohne Vorzeichen neuer Ablageort
//     (statt REAL nun DINT)
// 
//     3. Neue Ausgangsvariable Ready = Lesen/Schreiben der Parameter
//     abgeschlossen
// 
//     4. Austauch der Parameter kann jetzt abgebrochen werden
// 
//     5. Warnung durch Initialisierung elimininiert
// 
//     6. Eingang Laddr in hardwareId umbenannt
// 
// Änderung:  G.F. Typical Team                       24.11.16              4.5
//     - Fehlerausgabe bei unbekannten Datentyp (ErrorId := 5)
//     - Datentyp 10 (OctetString) wird unterstützt
//     - Datentyp 13 (TimeDifference) wird unterstützt
//     - Fehler bei Auftrag abbrechen behoben
// 
// Änderung:  G.F. Typical Team                       11.01.17              5.0
//     - Festlegung auf einheitlicher neuer Version 5.0 
// 
// Bibliothek V7
// Funktion: Austausch 15 beliebiger Parameter zwischen SINAMICS S120/G120 <-> S7
// ********************************************************************************************************************************************************
// ************************************************************************FB283***************************************************************************
// ********************************************************************************************************************************************************
   VAR_INPUT
      Start : Bool := 0;   // Start of the job (0 = no job or cancel the actual job; 1= start job and perform the job) / 0-->1 Start des gewählten azyklischen Auftrags
      ReadWrite : Bool := 0;   // Type of job 0 = read parameter, 1 = write parameter / 0 = Lesen; 1 = Schreiben
      ParaNo : Int := 1;   // Number of parameters to read or write / Anzahl der zu lesenden / schreibenden Parameter
      AxisNo : Byte := 16#01;   // Object ID of drive Output variables / Antriebsnummer
      hardwareId : Hw_Io := 0;   // Configured diagnosis address of the module (DEC) for WRREC and RDREC / Hardware Identifer des Modul Acces Points / Istwertslots des zyklsichen Telegramms
   END_VAR
   VAR_OUTPUT
      Ready : Bool := 0;   // Read or write parameter order ready / Bereitschaftsrückmeldung für den Betrieb mit LAcycCom Bausteinen
      Busy : Bool := 0;   // =1 Mode of operation is explained / 1 = Auftrag wird abgearbeitet
      Done : Bool := 1;   // =1 Mode of operation without mistake finishes / 1 = Auftrag wurde beendet
      Error : Bool := 0;   // Error or faults are active / 1 = Anzeige eines aufgetretenen Fehlers
      ErrorId : DWord := 0;   // Mode of operation disturbance / Binärcodierter Statusausgang (siehe Doku)
      DiagId : Word := 16#0000;   // Extended communication errorStatic variables / Rückmeldeausgang der Systemfunktionen im Fehlerfall
   END_VAR
   VAR
      sbWrError : Bool := 0;   // Error when writing with SFB WRREC
      sbWrDone : Bool := 0;   // Data record written with SFB WRREC
      sbRdError : Bool := 0;   // Error when reading with SFB RDREC
      sbWrBusy : Bool := 0;   // Write Task busy SFB 53 WRREC
      sbRdBusy : Bool := 0;   // Read Task busy SFB 52 RDREC
      sbWrStart : Bool := 0;   // Start write job
      sbRdStart : Bool := 0;   // Start read job
      sbWrStart1 : Bool := 0;   // Start write job (first part of write commando)
      sbRdStart1 : Bool := 0;   // Start read job (first part of read commando)
      sbWrStart2 : Bool := 0;   // Start write job (second part of write commando)
      sbRdStart2 : Bool := 0;   // Start read job (second part of read commando)
      sbStart : Bool := 0;   // Positive edge of Start commando
      sbReady : Bool := 0;   // Positive edge of Ready
      sbRead : Bool := 0;   // Commando "Read"
      sbWrite : Bool := 0;   // Commando "Write"
      sbParaNo : Bool := 0;   // The count of parameter are Okay
      sbBusy : Bool := 0;   // Mode of operation is explained
      sbError : Bool := 0;   // Error or faults are active
      sbDone : Bool := 0;   // Job finished
      siParaNo : Int := 0;   // Count of parameter are read or write
      syAxisNo : Byte := 0;   // Axis ID
      siReqRef : Int := 0;   // Reference number of request
      siErrorId : Int := 0;   // Function block fault ID
      siErrorCount : Int := 0;   // temporary error counter of retry job
      siMaxErrCount : Int := 12500;   // max. temporary error counter
      swParaError : Word := WORD#16#0000;   // Error of parameter
      sxReqParaMulti : Struct   // Telegramm for request/change parameter value, multi-parameter
         sxHeader : Struct   // Request header
            syReqRef : Byte := 16#00;   // Request reference (Request ID, mirrored in response)
            syReqId : Byte := 16#01;   // Request ID 0x1=Read
            syAxisNo : Byte := 16#00;   // Axis (0x0=Axis A | 0x1=Axis B)
            syParaNo : Byte := 16#00;   // No. of parameters (DEC: for single parameters=1)
         END_STRUCT;
         sxParaAdress : Array[1..16] of Struct   // Parameter address 1..16
            syAttr : Byte;   // Attribute of parameters (0x10=Value, 0x30=Text)
            syElemNo : Byte;   // No. of elements (DEC: for single elements=1)
            siParaNo : Int;   // Number of parameter (Number 1..65535)
            siIndex : Int;   // Subindex (Number 1..65535)
         END_STRUCT;
      END_STRUCT;
      sxChaParaMulti : Struct   // Telegramm for change parameter value, multi-parameter
         sxHeader : Struct   // Request header
            syReqRef : Byte := 16#00;   // Request reference (Request ID, mirrored in response)
            syReqId : Byte := 16#02;   // Request ID 0x2=Write
            syAxisNo : Byte := 16#00;   // Axis (0x0=Axis A | 0x1=Axis B)
            syParaNo : Byte := 16#00;   // No. of parameters (DEC: for single parameters=1)
         END_STRUCT;
         sxData : Array[1..192] of Byte;   // Parameter address 1..16 (Attribute/Value (BYTE), Number of Elements (BYTE), Parameter number (2 BYTES), Subindex (2 BYTES), Parameter value 1..16 (Format/Error (BYTE), Number of Values/Value of Error (BYTE), Value (BYTE or WORD or DWORD)
      END_STRUCT;
      sxRespParaMulti : Struct   // Telegramm for response parameter value, multi-parameter
         sxHeader : Struct   // Request header
            syReqRef : Byte := 16#00;   // Request reference (Request ID, mirrored in response)
            syReqId : Byte := 16#00;   // Request ID (0x1=Read | 0x2=Write)
            syAxisNo : Byte := 16#00;   // Axis (0x0=Axis A | 0x1=Axis B)
            syParaNo : Byte := 16#00;   // No. of parameters (DEC: for single parameters=1)
         END_STRUCT;
         sxData : Array[1..96] of Byte;   // Parameter value 1..16 (Format/Error (BYTE), Number of Values/Value of Error (BYTE), Value (BYTE or WORD or DWORD)
      END_STRUCT;
      sxParameter : Array[1..16] of Struct   // List of parameter (max. 16 parameter)
         siParaNo : Int;   // Number of parameter (Number 1..65535)
         siIndex : Int;   // Subindex (Number 1..65535)
         srValue : Real;   // Value of parameter
         sdValue : DInt;   // Value of parameter
         syFormat : Byte;   // Format of value (Format 0x40..0x44)
         swErrorNo : Word;   // Error number (see table below)
      END_STRUCT;
      RDREC_1 : RDREC;
      WRREC_1 : WRREC;
      siParaNoMax : Int := 16;   // max. Anzahl der Parameter
      siLenHeader : Int := 4;   // Length of telegram of header
      siLenParaMulti : Int := 96;   // Length of telegram of data for request and response
      siLenChaPara : Int := 192;   // Length of telegram of data for change parameterTemporary variables
   END_VAR
   VAR_TEMP
      piCount : Int;   // Freely available counter variable
      piPointer : Int;   // Freely available pointer array variable
      piLenTele : Int;   // Length of telegram of buffer
      piRetSFC : Int;   // Status for fault analysis
      pwWordHigh : Word;   // Help variable of word
      pwWordLow : Word;   // Help variable of word
      pwWord1 : Word;   // Help variable of word
      pwWord2 : Word;   // Help variable of word
      pdDWordHigh : DWord;   // Help variable of dword
      pdDWordLow : DWord;   // Help variable of dword
      pdStatus : DWord;   // Status[1] = Error => Status[2] Error Decode + Status[3] Error Code
      pbValidSFB : Bool;   // Status SFB
      piLenSFB : UInt;   // Status length for SFB call
      pwErrorNo : Word;   // Error number
   END_VAR
   // sxReqParaMulti.sxParaAdress[1].syAttr := 16#10;
   // sxReqParaMulti.sxParaAdress[2].syAttr := 16#10;
   // sxReqParaMulti.sxParaAdress[3].syAttr := 16#10;
   // sxReqParaMulti.sxParaAdress[4].syAttr := 16#10;
   // sxReqParaMulti.sxParaAdress[5].syAttr := 16#10;
   // sxReqParaMulti.sxParaAdress[6].syAttr := 16#10;
   // sxReqParaMulti.sxParaAdress[7].syAttr := 16#10;
   // sxReqParaMulti.sxParaAdress[8].syAttr := 16#10;
   // sxReqParaMulti.sxParaAdress[9].syAttr := 16#10;
   // sxReqParaMulti.sxParaAdress[10].syAttr := 16#10;
   // sxReqParaMulti.sxParaAdress[11].syAttr := 16#10;
   // sxReqParaMulti.sxParaAdress[12].syAttr := 16#10;
   // sxReqParaMulti.sxParaAdress[13].syAttr := 16#10;
   // sxReqParaMulti.sxParaAdress[14].syAttr := 16#10;
   // sxReqParaMulti.sxParaAdress[15].syAttr := 16#10;
   // sxReqParaMulti.sxParaAdress[16].syAttr := 16#10;
   // sxReqParaMulti.sxParaAdress[1].syElemNo := 16#01;
   // sxReqParaMulti.sxParaAdress[2].syElemNo := 16#01;
   // sxReqParaMulti.sxParaAdress[3].syElemNo := 16#01;
   // sxReqParaMulti.sxParaAdress[4].syElemNo := 16#01;
   // sxReqParaMulti.sxParaAdress[5].syElemNo := 16#01;
   // sxReqParaMulti.sxParaAdress[6].syElemNo := 16#01;
   // sxReqParaMulti.sxParaAdress[7].syElemNo := 16#01;
   // sxReqParaMulti.sxParaAdress[8].syElemNo := 16#01;
   // sxReqParaMulti.sxParaAdress[9].syElemNo := 16#01;
   // sxReqParaMulti.sxParaAdress[10].syElemNo := 16#01;
   // sxReqParaMulti.sxParaAdress[11].syElemNo := 16#01;
   // sxReqParaMulti.sxParaAdress[12].syElemNo := 16#01;
   // sxReqParaMulti.sxParaAdress[13].syElemNo := 16#01;
   // sxReqParaMulti.sxParaAdress[14].syElemNo := 16#01;
   // sxReqParaMulti.sxParaAdress[15].syElemNo := 16#01;
   // sxReqParaMulti.sxParaAdress[16].syElemNo := 16#01;
   // sxReqParaMulti.sxParaAdress[1].siParaNo := 0;
   // sxReqParaMulti.sxParaAdress[2].siParaNo := 0;
   // sxReqParaMulti.sxParaAdress[3].siParaNo := 0;
   // sxReqParaMulti.sxParaAdress[4].siParaNo := 0;
   // sxReqParaMulti.sxParaAdress[5].siParaNo := 0;
   // sxReqParaMulti.sxParaAdress[6].siParaNo := 0;
   // sxReqParaMulti.sxParaAdress[7].siParaNo := 0;
   // sxReqParaMulti.sxParaAdress[8].siParaNo := 0;
   // sxReqParaMulti.sxParaAdress[9].siParaNo := 0;
   // sxReqParaMulti.sxParaAdress[10].siParaNo := 0;
   // sxReqParaMulti.sxParaAdress[11].siParaNo := 0;
   // sxReqParaMulti.sxParaAdress[12].siParaNo := 0;
   // sxReqParaMulti.sxParaAdress[13].siParaNo := 0;
   // sxReqParaMulti.sxParaAdress[14].siParaNo := 0;
   // sxReqParaMulti.sxParaAdress[15].siParaNo := 0;
   // sxReqParaMulti.sxParaAdress[16].siParaNo := 0;
   // sxReqParaMulti.sxParaAdress[1].siIndex := 0;
   // sxReqParaMulti.sxParaAdress[2].siIndex := 0;
   // sxReqParaMulti.sxParaAdress[3].siIndex := 0;
   // sxReqParaMulti.sxParaAdress[4].siIndex := 0;
   // sxReqParaMulti.sxParaAdress[5].siIndex := 0;
   // sxReqParaMulti.sxParaAdress[6].siIndex := 0;
   // sxReqParaMulti.sxParaAdress[7].siIndex := 0;
   // sxReqParaMulti.sxParaAdress[8].siIndex := 0;
   // sxReqParaMulti.sxParaAdress[9].siIndex := 0;
   // sxReqParaMulti.sxParaAdress[10].siIndex := 0;
   // sxReqParaMulti.sxParaAdress[11].siIndex := 0;
   // sxReqParaMulti.sxParaAdress[12].siIndex := 0;
   // sxReqParaMulti.sxParaAdress[13].siIndex := 0;
   // sxReqParaMulti.sxParaAdress[14].siIndex := 0;
   // sxReqParaMulti.sxParaAdress[15].siIndex := 0;
   // sxReqParaMulti.sxParaAdress[16].siIndex := 0;
   // sxParameter[1].siParaNo := 0;
   // sxParameter[2].siParaNo := 0;
   // sxParameter[3].siParaNo := 0;
   // sxParameter[4].siParaNo := 0;
   // sxParameter[5].siParaNo := 0;
   // sxParameter[6].siParaNo := 0;
   // sxParameter[7].siParaNo := 0;
   // sxParameter[8].siParaNo := 0;
   // sxParameter[9].siParaNo := 0;
   // sxParameter[10].siParaNo := 0;
   // sxParameter[11].siParaNo := 0;
   // sxParameter[12].siParaNo := 0;
   // sxParameter[13].siParaNo := 0;
   // sxParameter[14].siParaNo := 0;
   // sxParameter[15].siParaNo := 0;
   // sxParameter[16].siParaNo := 0;
   // sxParameter[1].siIndex := 0;
   // sxParameter[2].siIndex := 0;
   // sxParameter[3].siIndex := 0;
   // sxParameter[4].siIndex := 0;
   // sxParameter[5].siIndex := 0;
   // sxParameter[6].siIndex := 0;
   // sxParameter[7].siIndex := 0;
   // sxParameter[8].siIndex := 0;
   // sxParameter[9].siIndex := 0;
   // sxParameter[10].siIndex := 0;
   // sxParameter[11].siIndex := 0;
   // sxParameter[12].siIndex := 0;
   // sxParameter[13].siIndex := 0;
   // sxParameter[14].siIndex := 0;
   // sxParameter[15].siIndex := 0;
   // sxParameter[16].siIndex := 0;
   // sxParameter[1].srValue := 0.0;
   // sxParameter[2].srValue := 0.0;
   // sxParameter[3].srValue := 0.0;
   // sxParameter[4].srValue := 0.0;
   // sxParameter[5].srValue := 0.0;
   // sxParameter[6].srValue := 0.0;
   // sxParameter[7].srValue := 0.0;
   // sxParameter[8].srValue := 0.0;
   // sxParameter[9].srValue := 0.0;
   // sxParameter[10].srValue := 0.0;
   // sxParameter[11].srValue := 0.0;
   // sxParameter[12].srValue := 0.0;
   // sxParameter[13].srValue := 0.0;
   // sxParameter[14].srValue := 0.0;
   // sxParameter[15].srValue := 0.0;
   // sxParameter[16].srValue := 0.0;
   // sxParameter[1].sdValue := 0;
   // sxParameter[2].sdValue := 0;
   // sxParameter[3].sdValue := 0;
   // sxParameter[4].sdValue := 0;
   // sxParameter[5].sdValue := 0;
   // sxParameter[6].sdValue := 0;
   // sxParameter[7].sdValue := 0;
   // sxParameter[8].sdValue := 0;
   // sxParameter[9].sdValue := 0;
   // sxParameter[10].sdValue := 0;
   // sxParameter[11].sdValue := 0;
   // sxParameter[12].sdValue := 0;
   // sxParameter[13].sdValue := 0;
   // sxParameter[14].sdValue := 0;
   // sxParameter[15].sdValue := 0;
   // sxParameter[16].sdValue := 0;
   // sxParameter[1].syFormat := BYTE#16#00;
   // sxParameter[2].syFormat := BYTE#16#00;
   // sxParameter[3].syFormat := BYTE#16#00;
   // sxParameter[4].syFormat := BYTE#16#00;
   // sxParameter[5].syFormat := BYTE#16#00;
   // sxParameter[6].syFormat := BYTE#16#00;
   // sxParameter[7].syFormat := BYTE#16#00;
   // sxParameter[8].syFormat := BYTE#16#00;
   // sxParameter[9].syFormat := BYTE#16#00;
   // sxParameter[10].syFormat := BYTE#16#00;
   // sxParameter[11].syFormat := BYTE#16#00;
   // sxParameter[12].syFormat := BYTE#16#00;
   // sxParameter[13].syFormat := BYTE#16#00;
   // sxParameter[14].syFormat := BYTE#16#00;
   // sxParameter[15].syFormat := BYTE#16#00;
   // sxParameter[16].syFormat := BYTE#16#00;
   // sxParameter[1].swErrorNo := WORD#16#0000;
   // sxParameter[2].swErrorNo := WORD#16#0000;
   // sxParameter[3].swErrorNo := WORD#16#0000;
   // sxParameter[4].swErrorNo := WORD#16#0000;
   // sxParameter[5].swErrorNo := WORD#16#0000;
   // sxParameter[6].swErrorNo := WORD#16#0000;
   // sxParameter[7].swErrorNo := WORD#16#0000;
   // sxParameter[8].swErrorNo := WORD#16#0000;
   // sxParameter[9].swErrorNo := WORD#16#0000;
   // sxParameter[10].swErrorNo := WORD#16#0000;
   // sxParameter[11].swErrorNo := WORD#16#0000;
   // sxParameter[12].swErrorNo := WORD#16#0000;
   // sxParameter[13].swErrorNo := WORD#16#0000;
   // sxParameter[14].swErrorNo := WORD#16#0000;
   // sxParameter[15].swErrorNo := WORD#16#0000;
   // sxParameter[16].swErrorNo := WORD#16#0000;
BEGIN

   //=============================================================================
   //SIEMENS AG
   //(c)Copyright 2017 All Rights Reserved
   //-----------------------------------------------------------------------------
   // Library: DriveLib
   // Tested with: S7-1516-3 PN/DP V1.8
   // Engineering: TIA Portal V14
   // Restrictions: -
   // Requirements: S7-1200 / S7-1500
   // Functionality: read and write up to 15 parameter from/to a Sinamics
   //
   //=============================================================================

   // Auftrag "Parameter lesen" bzw. Auftrag "Parameter schreiben" wird nicht mehr ausgeführt
   IF NOT #sbBusy THEN
     // Überprüfung der auf korrekte Parametrierung der Anzahl der Parameter
     IF #ParaNo > #siParaNoMax THEN

       #sbParaNo := FALSE;
       #sbError := True;
       #siErrorId := 2;
     ELSIF #ParaNo < 1 THEN

       #sbParaNo := FALSE;
       #sbError := True;
       #siErrorId := 2;
     ELSE

       #sbParaNo := TRUE;
       #siParaNo := #ParaNo;

       IF #siErrorId = 2 THEN
         #siErrorId := 0;
         #sbError := False;
       END_IF;
     END_IF;

     #syAxisNo := #AxisNo;
   END_IF;

   // Starten 
   IF #Start AND NOT #sbStart AND (#ParaNo <> 0) AND NOT #sbBusy THEN

     #sbReady := False;
     #sbError := False;
     #sbBusy := False;

     // Auftrag "Parameter lesen" erkennen
     IF NOT #ReadWrite THEN
       #sbRead := True;
       #sbWrStart := True;
       #sbRdStart := False;

       #sbWrite := False;
       #sbWrStart1 := False;
       #sbRdStart1 := False;
       #sbWrStart2 := False;
       #sbRdStart2 := False;

       // Referenzauftragsnummer erzeugen
       #siReqRef := #siReqRef + 1;

       // bei Überschreitung wieder zurücksetzen und von vorne (Wertebereich von 0-255)
       IF #siReqRef > 255 THEN
         #siReqRef := 0;
       END_IF;

       // Auftrag "Parameter schreiben" erkennen
     ELSE
       #sbWrite := True;
       #sbWrStart1 := True;
       #sbRdStart1 := False;
       #sbWrStart2 := False;
       #sbRdStart2 := False;

       #sbRead := False;
       #sbWrStart := False;
       #sbRdStart := False;

       // Referenzauftragsnummer erzeugen
       #siReqRef := #siReqRef + 1;

       // bei Überschreitung wieder zurücksetzen und von vorne (Wertebereich von 0-255)
       IF #siReqRef > 255 THEN
         #siReqRef := 0;
       END_IF;
     END_IF;

     // Fehler 4 und 5 wieder zurücknehmen
     IF (#siErrorId = 4) OR (#siErrorId = 5) THEN
       #sbError := False;
       #siErrorId := 0;
     END_IF;
   END_IF;

   // "Start commando" Flanke merken
   #sbStart := #Start;

   // Abbrechen
   IF NOT #Start THEN

     #siErrorCount := 0;
     // Schreib - oder Lesevorgang abbrechen
     #sbRead := False;
     #sbWrStart := False;
     #sbRdStart := False;

     #sbWrite := False;
     #sbWrStart1 := False;
     #sbRdStart1 := False;
     #sbWrStart2 := False;
     #sbRdStart2 := False;

     // Auftag ist noch beschäftigt => Fehler ausgeben
     IF #sbBusy THEN
       #sbError := True;
       #siErrorId := 4;
       #sbBusy := False;
     END_IF;
   END_IF;

   // Auftrag "Parameter lesen" wurde ausgelöst
   IF #sbParaNo AND #sbRead AND NOT #sbWrite THEN

     // Auftrag "Parameter lesen" vorbereiten und abschicken
     IF #sbWrStart THEN

       // Ablöschen des Sendepuffers
       IF NOT (#siParaNo = #siParaNoMax) THEN
         FOR #piCount := #siParaNo TO #siParaNoMax DO

           // Parameternummer des Parameters 
           #sxReqParaMulti.sxParaAdress[#piCount].siParaNo := 0;

           // Subindex des Parameters
           #sxReqParaMulti.sxParaAdress[#piCount].siIndex := 0;
         END_FOR;
       END_IF;

       // Auftrags-HEADER erstellen
       // Auftragsreferenz
       #sxReqParaMulti.sxHeader.syReqRef := INT_TO_BYTE(#siReqRef);

       // Auftragskennung 0x01=Request Parameters
       #sxReqParaMulti.sxHeader.syReqId := B#16#01;

       // Achse
       #sxReqParaMulti.sxHeader.syAxisNo := #syAxisNo;

       // Anzahl Parameter        
       #sxReqParaMulti.sxHeader.syParaNo := INT_TO_BYTE(#siParaNo);

       // Auftrags-PARAMETERADRESSE erstellen
       FOR #piCount := 1 TO #siParaNo DO

         // Parameternummer des Parameters                                
         #sxReqParaMulti.sxParaAdress[#piCount].siParaNo := #sxParameter[#piCount].siParaNo;

         // Subindex des Parameters
         #sxReqParaMulti.sxParaAdress[#piCount].siIndex := #sxParameter[#piCount].siIndex;
       END_FOR;

       // SCHREIBEN AZYKLISCH
       #piLenTele := #siLenHeader + #siLenParaMulti;
       #WRREC_1(REQ := True,                                // Startimpuls
                ID := #hardwareId,                         // Diagnoseadresse
                INDEX := 47,                                  // Rahmentyp
                LEN := INT_TO_UINT(#piLenTele),             // maximale Länge
                DONE => #sbWrDone,                           // Schreibauftrag beendet
                BUSY => #sbWrBusy,                           // Slave beschäftigt
                ERROR => #sbWrError,                          // Fehler beim Schreiben
                STATUS => #pdStatus,                           // Status[1] = Error => Status[2] Error Decode + Status[3] Error Code
                RECORD := #sxReqParaMulti);                    // Zeiger auf zu schreibenen Datensatzes

       // Ausgänge setzen
       #sbBusy := #sbWrBusy;
       #sbDone := #sbWrDone;

       // Fehler auswerten
       IF #sbWrError THEN

         // Fehlerstatus aus dem Doppelwort filtern und weitergeben                
         #pwWord1 := DWORD_TO_WORD(SHR(IN := (#pdStatus AND DW#16#FFFF00), N := 8));

         // Fehlerstatus setzen
         #siErrorId := 3;
         #DiagId := #pwWord1;

         //Temporärer Fehler: #pdStatus = 80A7, 80B5, 80C0, 80C1, 80C2, 80C3 oder 80C4 zulassen und nocheinmal versuchen
         IF NOT (#pwWord1 = DW#16#80A7) AND NOT (#pwWord1 = DW#16#80B5) AND NOT (#pwWord1 = DW#16#80C0) AND
           NOT (#pwWord1 = DW#16#80C1) AND NOT (#pwWord1 = DW#16#80C2) AND NOT (#pwWord1 = DW#16#80C3) AND
           NOT (#pwWord1 = DW#16#80C4) THEN

           // Wiederholungsauftrag wieder zurücknehmen 
           #sbWrStart := False;
           #sbRdStart := False;
           #sbRead := False;

           // Fehler ausgeben 
           #sbError := #sbWrError;

         ELSE
           // Fehlerwiederholauftrag ??                   
           IF #siErrorCount = #siMaxErrCount THEN

             // Wiederholungsauftrag wieder zurücknehmen
             #sbWrStart := False;
             #sbRdStart := False;
             #sbRead := False;

             //Fehlerzähler zurücksetzen
             #siErrorCount := 0;

             // Fehler ausgeben 
             #sbError := #sbWrError;

             // nix tun bis Zähler überläuft
           ELSE
             #siErrorCount := #siErrorCount + 1;
           END_IF;
         END_IF;

         // kein Fehler beim SCHEIBEN AZYKLISCH und Auftrag fertig 
       ELSIF NOT #sbWrBusy AND #sbWrDone THEN

         // Fehlerkennung zurücknehmen
         IF #siErrorId = 3 THEN
           #siErrorId := 0;
           #sbError := False;
         END_IF;

         #DiagId := W#16#00;

         // Schreibauftrag fertig melden und Leseantrag anstossen
         #sbWrStart := False;
         #sbRdStart := True;
       END_IF;
     END_IF; // Auftrag "Parameter lesen" vorbereiten und abschicken

     // vom Auftrag "Parameter lesen" die Antwort abwarten und dann auswerten
     IF #sbRdStart THEN

       // Ablöschen des Empfangspuffers
       #sxRespParaMulti.sxHeader.syReqRef := B#16#00;
       #sxRespParaMulti.sxHeader.syReqId := B#16#00;
       #sxRespParaMulti.sxHeader.syAxisNo := B#16#00;
       #sxRespParaMulti.sxHeader.syParaNo := B#16#00;

       FOR #piCount := 1 TO #siLenParaMulti DO
         #sxRespParaMulti.sxData[#piCount] := B#16#00;
       END_FOR;

       // LESEN AZYKLISCH
       #piLenTele := #siLenHeader + #siLenParaMulti;
       #RDREC_1(REQ := True,                                // Startimpuls
                ID := #hardwareId,                         // Diagnoseadresse        
                INDEX := 47,                                  // Rahmentyp           
                MLEN := INT_TO_UINT(#piLenTele),             // maximale Länge
                VALID => #pbValidSFB,                         // neuer Datensatz empfangen und gültig   
                BUSY => #sbRdBusy,                           // Slave beschäftigt
                ERROR => #sbRdError,                          // Fehler beim Schreiben
                STATUS => #pdStatus,                           // Status[1] = Error => Status[2] Error Decode + Status[3] Error Code 
                LEN => #piLenSFB,                           // Länge des gelesenen Datensatzes
                RECORD := #sxRespParaMulti);                   // Zeiger auf gelesenen Datensatz

       // Ausgänge setzen
       #sbBusy := #sbRdBusy;
       #sbDone := #pbValidSFB;

       // Fehler auswerten
       IF #sbRdError THEN
         // Fehlerstatus aus dem Doppelwort filtern und weitergeben                
         #pwWord1 := DWORD_TO_WORD(SHR(IN := (#pdStatus AND DW#16#FFFF00), N := 8));

         // Fehlerstatus setzen
         #siErrorId := 3;
         #DiagId := #pwWord1;

         //Temporärer Fehler: #pdStatus = 80A7, 80B5, 80C0, 80C1, 80C2, 80C3 oder 80C4 zulassen und nocheinmal versuchen
         IF NOT (#pwWord1 = DW#16#80A7) AND NOT (#pwWord1 = DW#16#80B5) AND NOT (#pwWord1 = DW#16#80C0) AND
           NOT (#pwWord1 = DW#16#80C1) AND NOT (#pwWord1 = DW#16#80C2) AND NOT (#pwWord1 = DW#16#80C3) AND
           NOT (#pwWord1 = DW#16#80C4) THEN

           // Wiederholungsauftrag wieder zurücknehmen  
           #sbWrStart := False;
           #sbRdStart := False;
           #sbRead := False;

           // Fehler ausgeben 
           #sbError := #sbRdError;

         ELSE
           // Fehlerwiederholauftrag ??                   
           IF #siErrorCount = #siMaxErrCount THEN

             // Wiederholungsauftrag wieder zurücknehmen
             #sbWrStart := False;
             #sbRdStart := False;
             #sbRead := False;

             //Fehlerzähler zurücksetzen
             #siErrorCount := 0;

             // Fehler ausgeben 
             #sbError := #sbRdError;

             // nix tun bis Zähler überläuft
           ELSE
             #siErrorCount := #siErrorCount + 1;
           END_IF;
         END_IF;

         // Fehler : die Auftragsreferenz der Antwort übertimmt nicht mit der Auftragsreferenz der Anfrage überein
       ELSIF NOT (#siReqRef = BYTE_TO_INT(#sxRespParaMulti.sxHeader.syReqRef)) AND NOT #sbRdBusy AND #pbValidSFB THEN
         #siErrorId := 1;
         #sbError := True;
         #sbDone := False;

         // Wiederholungsauftrag wieder zurücknehmen  
         #sbWrStart := False;
         #sbRdStart := False;
         #sbRead := False;

         // Fehler : falsche Auftragskennung zurück erhalten    
       ELSIF NOT (#sxRespParaMulti.sxHeader.syReqId = B#16#81 OR #sxRespParaMulti.sxHeader.syReqId = B#16#01) AND
         NOT #sbRdBusy AND #pbValidSFB THEN
         #siErrorId := 1;
         #sbError := True;
         #sbDone := False;

         // Wiederholungsauftrag wieder zurücknehmen  
         #sbWrStart := False;
         #sbRdStart := False;
         #sbRead := False;

         // Fehler : die angeforderte Anzahl Parameter entspricht nicht der übermittelten Anzahl Parameter überein
       ELSIF NOT (#siParaNo = BYTE_TO_INT(#sxRespParaMulti.sxHeader.syParaNo)) AND NOT #sbRdBusy AND #pbValidSFB THEN
         #siErrorId := 1;
         #sbError := True;
         #sbDone := False;

         // Wiederholungsauftrag wieder zurücknehmen  
         #sbWrStart := False;
         #sbRdStart := False;
         #sbRead := False;

         // Fehler : die Achse entspricht nicht der übergebenen Achse
       ELSIF NOT (#syAxisNo = #sxRespParaMulti.sxHeader.syAxisNo) AND NOT #sbRdBusy AND #pbValidSFB THEN
         #siErrorId := 1;
         #sbError := True;
         #sbDone := False;

         // Wiederholungsauftrag wieder zurücknehmen  
         #sbWrStart := False;
         #sbRdStart := False;
         #sbRead := False;

         // kein Fehler beim LESEN AZYKLISCH und Auftrag fertig 
       ELSIF NOT #sbRdBusy AND #pbValidSFB THEN

         // die angefragten Parameter auswerten und im Puffer abspeichern
         #piPointer := 1;
         #swParaError := 16#0;

         FOR #piCount := 1 TO #siParaNo DO

           // ermitteltes Format des Parameters abspeichern
           #sxParameter[#piCount].syFormat := #sxRespParaMulti.sxData[#piPointer];

           // Format = Error ? = > gesendeter Parameter fehlerhaft
           IF (BYTE_TO_INT(#sxRespParaMulti.sxData[#piPointer]) = 68) THEN

             // Format = Error, zwei Bytes zu übermittelten Fehlernummer zusammenfassen
             #pwWordHigh := SHL(IN := BYTE_TO_WORD(#sxRespParaMulti.sxData[#piPointer + 2]), N := 8);
             #pwWordLow := BYTE_TO_WORD(#sxRespParaMulti.sxData[#piPointer + 3]);

             #sbError := True;

             // ermittelte Fehlernummer im Puffer abspeichern
             #sxParameter[#piCount].swErrorNo := #pwWordHigh XOR #pwWordLow;

